10:
ProductionDataError_IndoPrint2:= CONCAT(ProductionData_IndoPrintError11.SERIALNOERROR,',');
ProductionDataError_IndoPrint2:=	 CONCAT( ProductionDataError_IndoPrint2,ProductionData_IndoPrintError11.SDATEERROR	);
ProductionDataError_IndoPrint2:= CONCAT( ProductionDataError_IndoPrint2,',');
(*ProductionDataError_IndoPrint2:=	 CONCAT( ProductionDataError_IndoPrint2,ProductionData_IndoPrintError11.STIMEEROOR);
ProductionDataError_IndoPrint2:= CONCAT( ProductionDataError_IndoPrint2,',');
ProductionDataError_IndoPrint2:=	 CONCAT( ProductionDataError_IndoPrint2,ProductionData_IndoPrintError11.SHIFTERROR	);
ProductionDataError_IndoPrint2:= CONCAT( ProductionDataError_IndoPrint2,',');*)
ProductionDataError_IndoPrint2:=	 CONCAT( ProductionDataError_IndoPrint2,ProductionData_IndoPrintError11.ERRORIDERROR);
ProductionDataError_IndoPrint2:= CONCAT( ProductionDataError_IndoPrint2,'$0A');
(*ProductionData_IndoPrint2:=	 CONCAT( ProductionData_IndoPrint2,ProductionData_IndoPrint11.LOTNO);
ProductionData_IndoPrint2:= CONCAT( ProductionData_IndoPrint2,',');
ProductionData_IndoPrint2:=	 CONCAT( ProductionData_IndoPrint2,ProductionData_IndoPrint11.DFLTNETWEIGHT);
ProductionData_IndoPrint2:= CONCAT( ProductionData_IndoPrint2,',');
ProductionData_IndoPrint2:=	 CONCAT( ProductionData_IndoPrint2,ProductionData_IndoPrint11.ACTNETWEIGHT);
ProductionData_IndoPrint2:= CONCAT( ProductionData_IndoPrint2,'$0A');
ProductionData_IndoPrint2:=	 CONCAT( ProductionData_IndoPrint2,ProductionData_IndoPrint11.DFLTGROSSWEIGHT);
ProductionData_IndoPrint2:= CONCAT( ProductionData_IndoPrint2,',');
ProductionData_IndoPrint2:=	 CONCAT( ProductionData_IndoPrint2,ProductionData_IndoPrint11.ACTGROSSWEIGHT);
ProductionData_IndoPrint2:= CONCAT( ProductionData_IndoPrint2,'$0A');
ProductionData_IndoPrint2:=	 CONCAT( ProductionData_IndoPrint2,ProductionData_IndoPrint11.NetWt9);
ProductionData_IndoPrint2:= CONCAT( ProductionData_IndoPrint2,',');
ProductionData_IndoPrint2:=	 CONCAT( ProductionData_IndoPrint2,ProductionData_IndoPrint11.NetWt10);
ProductionData_IndoPrint2:= CONCAT( ProductionData_IndoPrint2,',');
ProductionData_IndoPrint2:=	 CONCAT( ProductionData_IndoPrint2,ProductionData_IndoPrint11.NetWt11);
ProductionData_IndoPrint2:= CONCAT( ProductionData_IndoPrint2,',');
ProductionData_IndoPrint2:=	 CONCAT( ProductionData_IndoPrint2,ProductionData_IndoPrint11.NetWt12);
ProductionData_IndoPrint2:= CONCAT( ProductionData_IndoPrint2,',');*)
ReportBot1Error_Indo:=FALSE;ReportSaveErrror:=FALSE;
IndoReport:=15;


11:	ProductionDataValuesError_IndoPrint_Com:=ProductionDataError_IndoPrint2;
TON_Indo3(IN:=TRUE , PT:=t#5s , Q=> , ET=> );
	FB_FileWrite_Indo.bExecute:=TRUE;
	IF NOT FB_FileWrite_Indo.bBusy AND NOT FB_FileWrite_Indo.bError AND TON_Indo3.Q THEN IndoReport:=IndoReport+1; END_IF

12:	FB_FileWrite_Indo.bExecute:=FALSE;(*ProductionData_IndoPrint:='';*)IndoReport:=IndoReport+1;

13:	ReportBot2Error_Indo:=TRUE;
	IF ReportBot2Error_Indo THEN IndoReport:=IndoReport+1;END_IF

14:(*	ProductionData_IndoPrint2:= CONCAT(ProductionData_IndoPrint11.NetWt13,',');
ProductionData_IndoPrint2:=	 CONCAT( ProductionData_IndoPrint2,ProductionData_IndoPrint11.NetWt14	);
ProductionData_IndoPrint2:= CONCAT( ProductionData_IndoPrint2,',');
ProductionData_IndoPrint2:=	 CONCAT( ProductionData_IndoPrint2,ProductionData_IndoPrint11.NetWt15);
ProductionData_IndoPrint2:= CONCAT( ProductionData_IndoPrint2,',');
ProductionData_IndoPrint2:=	 CONCAT( ProductionData_IndoPrint2,ProductionData_IndoPrint11.NetWt16);
ProductionData_IndoPrint2:= CONCAT( ProductionData_IndoPrint2,',');
ProductionData_IndoPrint2:=	 CONCAT( ProductionData_IndoPrint2,ProductionData_IndoPrint11.NetWt17);
ProductionData_IndoPrint2:= CONCAT( ProductionData_IndoPrint2,',');
ProductionData_IndoPrint2:=	 CONCAT( ProductionData_IndoPrint2,ProductionData_IndoPrint11.NetWt18);
ProductionData_IndoPrint2:= CONCAT( ProductionData_IndoPrint2,',');
ProductionData_IndoPrint2:=	 CONCAT( ProductionData_IndoPrint2,ProductionData_IndoPrint11.NetWt19);
ProductionData_IndoPrint2:= CONCAT( ProductionData_IndoPrint2,',');
ProductionData_IndoPrint2:=	 CONCAT( ProductionData_IndoPrint2,ProductionData_IndoPrint11.NetWt20);
ProductionData_IndoPrint2:= CONCAT( ProductionData_IndoPrint2,',');
ProductionData_IndoPrint2:=	 CONCAT( ProductionData_IndoPrint2,ProductionData_IndoPrint11.NetWt21);
ProductionData_IndoPrint2:= CONCAT( ProductionData_IndoPrint2,',');
ProductionData_IndoPrint2:=	 CONCAT( ProductionData_IndoPrint2,ProductionData_IndoPrint11.NetWt22);
ProductionData_IndoPrint2:= CONCAT( ProductionData_IndoPrint2,',');
ProductionData_IndoPrint2:=	 CONCAT( ProductionData_IndoPrint2,ProductionData_IndoPrint11.NetWt23);
ProductionData_IndoPrint2:= CONCAT( ProductionData_IndoPrint2,',');
ProductionData_IndoPrint2:=	 CONCAT( ProductionData_IndoPrint2,ProductionData_IndoPrint11.NetWt24);
ProductionData_IndoPrint2:= CONCAT( ProductionData_IndoPrint2,'$0A');*)
ReportBot2Error_Indo:=FALSE;
IndoReport:=IndoReport+1;

15:ProductionDataValuesError_IndoPrint_Com:=ProductionDataError_IndoPrint2;
TON_Indo4(IN:=TRUE , PT:=t#5s , Q=> , ET=> );

	FB_FileWrite_Indo.bExecute:=TRUE; IndoReport:=IndoReport+1;
	(*IF NOT FB_FileWrite_Indo.bBusy AND NOT FB_FileWrite_Indo.bError AND TON_Indo4.Q  THEN IndoReport:=IndoReport+1;END_IF*)

16:	IF NOT FB_FileWrite_Indo.bBusy AND NOT FB_FileWrite_Indo.bError (*AND TON_Indo4.Q*)  THEN FB_FileWrite_Indo.bExecute:=FALSE; IndoReport:=IndoReport+1;END_IF


17:	TON_Indo3(IN:=FALSE);TON_Indo4(IN:=FALSE);TON_Indo2(IN:=FALSE);TON_Indo1(IN:=FALSE);FB_FileWrite_Indo.bExecute:=FALSE;IndoReport:=IndoReport+1;

18:	FB_FileClose_Indo.bExecute:=TRUE;
	 IF NOT FB_FileClose_Indo.bBusy AND NOT FB_FileClose_Indo.bError THEN  IndoReport:=20;END_IF

19:	IF bANewDayError THEN IndoReport:=IndoReport+1;
	ELSIF NOT bANewDayError THEN FB_FileOpen_Indo.bExecute:=FALSE; IndoReport:=9;
END_IF

20:	FB_FileOpen_Indo.bExecute:=FALSE;SerialNoError:=SerialNoError+1;IndoReport:=9;

END_CASE

R_TRIG_ErrorRepo_Int(CLK:=bInitializeHmi , Q=> );

IF sDay <> sOldDayError THEN bANewDayError:=TRUE;IndoReport:=0; END_IF
TON_NEWDAYError(IN:=bANewDayError , PT:=T#0.5s , Q=> , ET=> );



CASE WriteError OF
0:	IF FB_FileWrite_Indo.bError THEN FB_FileWrite_Indo.bExecute:=FALSE;TON_writedly(IN:=FALSE);
	WriteError:=WriteError+1;END_IF

1:	TON_writedly(IN:=TRUE , PT:=t#2s , Q=> , ET=> );
	IF TON_writedly.Q THEN FB_FileWrite_Indo.bExecute:=TRUE;WriteError:=WriteError+1;END_IF

2:	TON_writedly(IN:=FALSE);WriteError:=0;

END_CASE




CASE OpenError OF


0:	IF FB_FileWrite_Indo.bError THEN FB_FileWrite_Indo.bExecute:=FALSE;TON_Opendly(IN:=FALSE);
	OpenError:=OpenError+1;END_IF

1:	TON_Opendly(IN:=TRUE , PT:=t#2s , Q=> , ET=> );
	IF TON_Opendly.Q THEN FB_FileWrite_Indo.bExecute:=TRUE;OpenError:=OpenError+1;END_IF

2:	TON_Opendly(IN:=FALSE);OpenError:=0;

END_CASE









		ProductionData_IndoPrintError11.SERIALNOERROR	:=DINT_TO_STRING(SerialNoError);
		ProductionData_IndoPrintError11.SDATEERROR	:=(sTIME);
		(*ProductionData_IndoPrintError11.SHIFTERROR	:=(sShitToReport);*)
		ProductionData_IndoPrintError11.ERRORIDERROR	:=(AlarmData);
		(*ProductionData_IndoPrint11.LOTNO	:=(LOTNO_DIS);
		ProductionData_IndoPrint11.DFLTNETWEIGHT	:=(Default_NetWeight_Report);
		ProductionData_IndoPrint11.ACTNETWEIGHT	:=(Actual_NetWeight_Report);
		ProductionData_IndoPrint11.DFLTGROSSWEIGHT	:=(Default_GrossWeight_Report);
		ProductionData_IndoPrint11.ACTGROSSWEIGHT	:=(Actual_GrossWeight_Report);
		ProductionData_IndoPrint11.NetWt9	:=REAL_TO_STRING(Cone_9_Wt);
		ProductionData_IndoPrint11.NetWt10	:=REAL_TO_STRING(Cone_10_Wt);
		ProductionData_IndoPrint11.NetWt11	:=REAL_TO_STRING(Cone_11_Wt);
		ProductionData_IndoPrint11.NetWt12	:=REAL_TO_STRING(Cone_12_Wt);
		ProductionData_IndoPrint11.NetWt13	:=REAL_TO_STRING(Cone_13_Wt);
		ProductionData_IndoPrint11.NetWt14	:=REAL_TO_STRING(Cone_14_Wt);
		ProductionData_IndoPrint11.NetWt15	:=REAL_TO_STRING(Cone_15_Wt);
		ProductionData_IndoPrint11.NetWt16	:=REAL_TO_STRING(Cone_16_Wt);
		ProductionData_IndoPrint11.NetWt17	:=REAL_TO_STRING(Cone_17_Wt);
		ProductionData_IndoPrint11.NetWt18	:=REAL_TO_STRING(Cone_18_Wt);
		ProductionData_IndoPrint11.NetWt19	:=REAL_TO_STRING(Cone_19_Wt);
		ProductionData_IndoPrint11.NetWt20	:=REAL_TO_STRING(Cone_20_Wt);
		ProductionData_IndoPrint11.NetWt21	:=REAL_TO_STRING(Cone_21_Wt);
		ProductionData_IndoPrint11.NetWt22	:=REAL_TO_STRING(Cone_22_Wt);
		ProductionData_IndoPrint11.NetWt23	:=REAL_TO_STRING(Cone_23_Wt);
		ProductionData_IndoPrint11.NetWt24	:=REAL_TO_STRING(Cone_24_Wt);*)
END_PROGRAM

(* POU Date_Time, ST *)
PROGRAM Date_Time
VAR
	ReportPath: STRING;



	sDayF1: STRING;
	sMonthF1: STRING;
	sDayMonth1: STRING;

END_VAR
				(****************REPORT DATA***********)
IF DfltWtPrint THEN NetwtPrint:=Default_NetWeight_Report;
ELSIF NOT DfltWtPrint THEN NetwtPrint:=Actual_NetWeight_Report;END_IF

IF GrossWtPrintDflt THEN GrosswtPrint:=Default_GrossWeight_Report;
ELSE GrosswtPrint:=Actual_GrossWeight_Report;END_IF



Actual_NetWeight_Report:=MID(STR:=REAL_TO_STRING(var_5), LEN:=6, POS:=1);
Default_NetWeight_Report:=MID(STR:=REAL_TO_STRING(DefaultNetWt), LEN:=6, POS:=1);

Actual_GrossWeight_Report:=MID(STR:=REAL_TO_STRING(rGrossWeight), LEN:=6, POS:=1);
Default_GrossWeight_Report:=MID(STR:=REAL_TO_STRING(DefaultGrossWt), LEN:=6, POS:=1);




					(****************DATE AND TIME***********)

(*======================= RTC==============================*)

FB_DateTime_1(NET_ID:='5.69.203.190.1.1 ' , Date_Time=> );

IF FB_DateTime_1.FBLTIME.systemTime.wHour >0 AND  FB_DateTime_1.FBLTIME.systemTime.wHour<9 THEN sHourPreFix:='0';

sHou:=CONCAT(STR1:=sHourPreFix, Str2:=WORD_TO_STRING(FB_DateTime_1.FBLTIME.systemTime.wHour));

ELSIF FB_DateTime_1.FBLTIME.systemTime.wHour >=10 AND  FB_DateTime_1.FBLTIME.systemTime.wHour<=24 THEN

sHou:=WORD_TO_STRING(FB_DateTime_1.FBLTIME.systemTime.wHour);

END_IF




IF FB_DateTime_1.FBLTIME.systemTime.wDay >0 AND  FB_DateTime_1.FBLTIME.systemTime.wDay<10 THEN sDayPreFix:='0';

sDay:=CONCAT(STR1:=sDayPreFix, Str2:=WORD_TO_STRING(FB_DateTime_1.FBLTIME.systemTime.wDay));

ELSIF FB_DateTime_1.FBLTIME.systemTime.wDay >=10 AND  FB_DateTime_1.FBLTIME.systemTime.wDay<=31 THEN

sDay:=WORD_TO_STRING(FB_DateTime_1.FBLTIME.systemTime.wDay);

END_IF




IF FB_DateTime_1.FBLTIME.systemTime.wMonth >0 AND  FB_DateTime_1.FBLTIME.systemTime.wMonth<10 THEN sMonthPreFix:='0';

sMonth:=CONCAT(STR1:=sMonthPreFix, Str2:=WORD_TO_STRING(FB_DateTime_1.FBLTIME.systemTime.wMonth));

ELSIF FB_DateTime_1.FBLTIME.systemTime.wMonth >=10 AND  FB_DateTime_1.FBLTIME.systemTime.wMonth<=12 THEN

sMonth:=WORD_TO_STRING(FB_DateTime_1.FBLTIME.systemTime.wMonth);

END_IF



sDayF1:=CONCAT(STR1:=sDay, STR2:=':');
sMonthF1:=CONCAT(STR1:=sMonth, STR2:=':');
sDayMonth1:=CONCAT(STR1:=sDayF1, STR2:=sMonthF1);
sDayMonthYear1:=CONCAT(STR1:=sDayMonth1, STR2:=WORD_TO_STRING(FB_DateTime_1.FBLTIME.systemTime.wYear));


sDaateReport:=(sDayMonthYear1);





sDayF:=CONCAT(STR1:=sDay, STR2:='_');
sMonthF:=CONCAT(STR1:=sMonth, STR2:='_');
sDayMonth:=CONCAT(STR1:=sDayF, STR2:=sMonthF);
sDayMonthYear:=CONCAT(STR1:=sDayMonth, STR2:=WORD_TO_STRING(FB_DateTime_1.FBLTIME.systemTime.wYear));

ReportPath:=CONCAT(STR1:='ProductionData', STR2:='_');
ReportPath_Final:=CONCAT(STR1:=ReportPath, STR2:=sDayMonthYear);

ReportPath_Final_1:=CONCAT(STR1:='\\ACP\Reports\', STR2:=ReportPath_Final);
ReportPath_Final_2:=CONCAT(STR1:=ReportPath_Final_1, STR2:='.csv');





sDayF1:=CONCAT(STR1:=sDay, STR2:=':');
sMonthF1:=CONCAT(STR1:=sMonth, STR2:=':');
sDayMonth1:=CONCAT(STR1:=sDayF1, STR2:=sMonthF1);
sDayMonthYear1:=CONCAT(STR1:=sDayMonth1, STR2:=WORD_TO_STRING(FB_DateTime_1.FBLTIME.systemTime.wYear));


sDaateReport:=(sDayMonthYear1);





sDayF:=CONCAT(STR1:=sDay, STR2:='_');
sMonthF:=CONCAT(STR1:=sMonth, STR2:='_');
sDayMonth:=CONCAT(STR1:=sDayF, STR2:=sMonthF);
sDayMonthYear:=CONCAT(STR1:=sDayMonth, STR2:=WORD_TO_STRING(FB_DateTime_1.FBLTIME.systemTime.wYear));

ReportPathError:=CONCAT(STR1:='ErrorData', STR2:='_');
ReportPath_FinalError:=CONCAT(STR1:=ReportPathError, STR2:=sDayMonthYear);

ReportPath_Final_1Error:=CONCAT(STR1:='\\ACP\Reports\', STR2:=ReportPath_FinalError);
ReportPath_Final_2Error:=CONCAT(STR1:=ReportPath_Final_1Error, STR2:='.csv');








DateTimeVar:=FB_DateTime_1.Date_Time;
END_PROGRAM

(* POU Parameters, ST *)
PROGRAM Parameters
VAR
	R_TRIG_1: R_TRIG;

	PrintVar: INT;




	ItemCodeHm21: BOOL;
END_VAR
IF SAVE AND PRGNO=1 AND NegTolEnableHmi THEN NegTol1:=1;ELSIF SAVE AND PRGNO=1 AND NOT  NegTolEnableHmi THEN  NegTol1:=0;END_IF
IF SAVE AND PRGNO=2 AND NegTolEnableHmi THEN NegTol2:=1;ELSIF SAVE AND PRGNO=2 AND NOT NegTolEnableHmi THEN  NegTol2:=0;END_IF
IF SAVE AND PRGNO=3 AND NegTolEnableHmi THEN NegTol3:=1;ELSIF SAVE AND PRGNO=3 AND NOT NegTolEnableHmi THEN  NegTol3:=0;END_IF
IF SAVE AND PRGNO=4 AND NegTolEnableHmi THEN NegTol4:=1;ELSIF SAVE AND PRGNO=4 AND NOT NegTolEnableHmi THEN  NegTol4:=0;END_IF
IF SAVE AND PRGNO=5 AND NegTolEnableHmi THEN NegTol5:=1;ELSIF SAVE AND PRGNO=5 AND NOT NegTolEnableHmi THEN  NegTol5:=0;END_IF

IF SAVE AND PRGNO=1 THEN

	PRGNO1:=PRGNO;
	COUNT1:=COUNT;
	CARTONNO1:=CARTONNO;
	DFLTNETWT1:=DFLTNETWT;
	DFLTGROSSWT1:=DFLTGROSSWT;
	BLEND1:=BLEND;
	SHADE1:=SHADE;
	CONETIP1:=CONETIP;
	CONELENGTH1:=CONELENGTH;
	CONENETWT1:=CONENETWT;
	NOOFCONES1:=NOOFCONES;
	LOTNO1:=LOTNO;
	WORKORDERNO1:=WORKORDERNO;
	NETWTTOL1:=NETWTTOL;
	GROSSWTTOL1:=GROSSWTTOL;
	DOM_EXPORT1:=DOM_EXPORT;
	PACKTYPE1:=PACKTYPE;

	ItemCodeHmi1:=ItemCodeHmi;
	IssueDesp1:=IssueDesp;
	Location1:=Location;
	Description1:=Description;
	Remarks1:=Remarks;
	Fyear1:=Fyear;
	AvgCount1:=AvgCount;
	TareWeight1:=TareWeight;
	BarCode1:=BarCode;
	WorkFlag1:=WorkFlag;
	EmptyConeWt1:=EmptyConeWt;


ELSIF SAVE AND PRGNO=2 THEN

	PRGNO2:=PRGNO;
	COUNT2:=COUNT;
	CARTONNO2:=CARTONNO;
	DFLTNETWT2:=DFLTNETWT;
	DFLTGROSSWT2:=DFLTGROSSWT;
	BLEND2:=BLEND;
	SHADE2:=SHADE;
	CONETIP2:=CONETIP;
	CONELENGTH2:=CONELENGTH;
	CONENETWT2:=CONENETWT;
	NOOFCONES2:=NOOFCONES;
	LOTNO2:=LOTNO;
	WORKORDERNO2:=WORKORDERNO;
	NETWTTOL2:=NETWTTOL;
	GROSSWTTOL2:=GROSSWTTOL;
	DOM_EXPORT2:=DOM_EXPORT;
	PACKTYPE2:=PACKTYPE;

	ItemCodeHmI2:=ItemCodeHmi;
	IssueDesp2:=IssueDesp;
	Location2:=Location;
	Description2:=Description;
	Remarks2:=Remarks;
	Fyear2:=Fyear;
	AvgCount2:=AvgCount;
	TareWeight2:=TareWeight;
	BarCode2:=BarCode;
	WorkFlag2:=WorkFlag;
	EmptyConeWt2:=EmptyConeWt;

ELSIF SAVE AND PRGNO=3 THEN

	PRGNO3:=PRGNO;
	COUNT3:=COUNT;
	CARTONNO3:=CARTONNO;
	DFLTNETWT3:=DFLTNETWT;
	DFLTGROSSWT3:=DFLTGROSSWT;
	BLEND3:=BLEND;
	SHADE3:=SHADE;
	CONETIP3:=CONETIP;
	CONELENGTH3:=CONELENGTH;
	CONENETWT3:=CONENETWT;
	NOOFCONES3:=NOOFCONES;
	LOTNO3:=LOTNO;
	WORKORDERNO3:=WORKORDERNO;
	NETWTTOL3:=NETWTTOL;
	GROSSWTTOL3:=GROSSWTTOL;
	DOM_EXPORT3:=DOM_EXPORT;
	PACKTYPE3:=PACKTYPE;

ItemCodeHmI3:=ItemCodeHmi;
	IssueDesp3:=IssueDesp;
	Location3:=Location;
	Description3:=Description;
	Remarks3:=Remarks;
	Fyear3:=Fyear;
	AvgCount3:=AvgCount;
	TareWeight3:=TareWeight;
	BarCode3:=BarCode;
	WorkFlag3:=WorkFlag;
	EmptyConeWt3:=EmptyConeWt;


ELSIF SAVE AND PRGNO=4 THEN

	PRGNO4:=PRGNO;
	COUNT4:=COUNT;
	CARTONNO4:=CARTONNO;
	DFLTNETWT4:=DFLTNETWT;
	DFLTGROSSWT4:=DFLTGROSSWT;
	BLEND4:=BLEND;
	SHADE4:=SHADE;
	CONETIP4:=CONETIP;
	CONELENGTH4:=CONELENGTH;
	CONENETWT4:=CONENETWT;
	NOOFCONES4:=NOOFCONES;
	LOTNO4:=LOTNO;
	WORKORDERNO4:=WORKORDERNO;
	NETWTTOL4:=NETWTTOL;
	GROSSWTTOL4:=GROSSWTTOL;
	DOM_EXPORT4:=DOM_EXPORT;
	PACKTYPE4:=PACKTYPE;

ItemCodeHmI4:=ItemCodeHmi;
	IssueDesp4:=IssueDesp;
	Location4:=Location;
	Description4:=Description;
	Remarks4:=Remarks;
	Fyear4:=Fyear;
	AvgCount4:=AvgCount;
	TareWeight4:=TareWeight;
	BarCode4:=BarCode;
	WorkFlag4:=WorkFlag;
	EmptyConeWt4:=EmptyConeWt;

ELSIF SAVE AND PRGNO=5 THEN

	PRGNO5:=PRGNO;
	COUNT5:=COUNT;
	CARTONNO5:=CARTONNO;
	DFLTNETWT5:=DFLTNETWT;
	DFLTGROSSWT5:=DFLTGROSSWT;
	BLEND5:=BLEND;
	SHADE5:=SHADE;
	CONETIP5:=CONETIP;
	CONELENGTH5:=CONELENGTH;
	CONENETWT5:=CONENETWT;
	NOOFCONES5:=NOOFCONES;
	LOTNO5:=LOTNO;
	WORKORDERNO5:=WORKORDERNO;
	NETWTTOL5:=NETWTTOL;
	GROSSWTTOL5:=GROSSWTTOL;
	DOM_EXPORT5:=DOM_EXPORT;
	PACKTYPE5:=PACKTYPE;

	ItemCodeHmI5:=ItemCodeHmi;
	IssueDesp5:=IssueDesp;
	Location5:=Location;
	Description5:=Description;
	Remarks5:=Remarks;
	Fyear5:=Fyear;
	AvgCount5:=AvgCount;
	TareWeight5:=TareWeight;
	BarCode5:=BarCode;
	WorkFlag5:=WorkFlag;
	EmptyConeWt5:=EmptyConeWt;

ELSIF SAVE AND PRGNO=6 THEN

	PRGNO6:=PRGNO;
	COUNT6:=COUNT;
	DETAILS6:=DETAILS;
	LOTNO6:=LOTNO;
	CARTONNO6:=CARTONNO;
	WORKORDERNO6:=WORKORDERNO;
	BLEND6:=BLEND;
	SHADE6:=SHADE;
	CONETIP6:=CONETIP;
	CONELENGTH6:=CONELENGTH;
	CONENETWT6:=CONENETWT;
	DFLTNETWT6:=DFLTNETWT;
	NETWTTOL6:=NETWTTOL;
	DFLTGROSSWT6:=DFLTGROSSWT;
	GROSSWTTOL6:=GROSSWTTOL;


ELSIF SAVE AND PRGNO=7 THEN

	PRGNO7:=PRGNO;
	COUNT7:=COUNT;
	DETAILS7:=DETAILS;
	LOTNO7:=LOTNO;
	CARTONNO7:=CARTONNO;
	WORKORDERNO7:=WORKORDERNO;
	BLEND7:=BLEND;
	SHADE7:=SHADE;
	CONETIP7:=CONETIP;
	CONELENGTH7:=CONELENGTH;
	CONENETWT7:=CONENETWT;
	DFLTNETWT7:=DFLTNETWT;
	NETWTTOL7:=NETWTTOL;
	DFLTGROSSWT7:=DFLTGROSSWT;
	GROSSWTTOL7:=GROSSWTTOL;


ELSIF SAVE AND PRGNO=8 THEN

	PRGNO8:=PRGNO;
	COUNT8:=COUNT;
	DETAILS8:=DETAILS;
	LOTNO8:=LOTNO;
	CARTONNO8:=CARTONNO;
	WORKORDERNO8:=WORKORDERNO;
	BLEND8:=BLEND;
	SHADE8:=SHADE;
	CONETIP8:=CONETIP;
	CONELENGTH8:=CONELENGTH;
	CONENETWT8:=CONENETWT;
	DFLTNETWT8:=DFLTNETWT;
	NETWTTOL8:=NETWTTOL;
	DFLTGROSSWT8:=DFLTGROSSWT;
	GROSSWTTOL8:=GROSSWTTOL;


ELSIF SAVE AND PRGNO=9 THEN

	PRGNO9:=PRGNO;
	COUNT9:=COUNT;
	DETAILS9:=DETAILS;
	LOTNO9:=LOTNO;
	CARTONNO9:=CARTONNO;
	WORKORDERNO9 :=WORKORDERNO;
	BLEND9 :=BLEND;
	SHADE9 :=SHADE;
	CONETIP9 :=CONETIP;
	CONELENGTH9 :=CONELENGTH;
	CONENETWT9 :=CONENETWT;
	DFLTNETWT9 :=DFLTNETWT;
	NETWTTOL9 :=NETWTTOL;
	DFLTGROSSWT9 :=DFLTGROSSWT;
	GROSSWTTOL9 :=GROSSWTTOL;


ELSIF SAVE AND PRGNO=10 THEN

	PRGNO10:=PRGNO;
	COUNT10:=COUNT;
	DETAILS10:=DETAILS;
	LOTNO10:=LOTNO;
	CARTONNO10:=CARTONNO;
	WORKORDERNO10:=WORKORDERNO;
	BLEND10:=BLEND;
	SHADE10:=SHADE;
	CONETIP10:=CONETIP;
	CONELENGTH10:=CONELENGTH;
	CONENETWT10:=CONENETWT;
	DFLTNETWT10:=DFLTNETWT;
	NETWTTOL10:=NETWTTOL;
	DFLTGROSSWT10:=DFLTGROSSWT;
	GROSSWTTOL10:=GROSSWTTOL;

END_IF










IF LOAD AND PRGNO_LOAD=1 THEN


	PRGNO_DIS:=PRGNO1;
	COUNT_DIS:=COUNT1;
	CARTONNO_DIS:=CARTONNO1;
	DFLTNETWT_DIS:=DFLTNETWT1;
	DFLTGROSSWT_DIS:=DFLTGROSSWT1;
	BLEND_DIS:=BLEND1;
	SHADE_DIS:=SHADE1;
	CONETIP_DIS:=CONETIP1;
	CONELENGTH_DIS:=CONELENGTH1;
	CONENETWT_DIS:=CONENETWT1;
	NOOFCONES_DIS:=NOOFCONES1;
	LOTNO_DIS:=LOTNO1;
	WORKORDERNO_DIS:=WORKORDERNO1;
	NETWTTOL_DIS:=NETWTTOL1;
	GROSSWTTOL_DIS:=GROSSWTTOL1;
	DOM_EXPORT_DIS:=DOM_EXPORT1;
	PACKTYPE_DIS:=PACKTYPE1;
	NegTol_DIS:=NegTol1;
	PRG1RUNNING:=TRUE;
	PRG2RUNNING:=FALSE;
	PRG3RUNNING:=FALSE;
	PRG4RUNNING:=FALSE;
	PRG5RUNNING:=FALSE;
	PRG6RUNNING:=FALSE;
	PRG7RUNNING:=FALSE;
	PRG8RUNNING:=FALSE;
	PRG9RUNNING:=FALSE;
	PRG10RUNNING:=FALSE;


ItemCodeHmi_DIS:=ItemCodeHmi1;
IssueDesp_DIS:=	IssueDesp1;
Location_DIS:=Location1;
Description_DIS:=	Description1;
Remarks_DIS:=	Remarks1;
Fyear_DIS:=	Fyear1;
AvgCount_DIS:=	AvgCount1;
TareWeight_DIS:=	TareWeight1;
BarCode_DIS:=	BarCode1;
WorkFlag_DIS:=	WorkFlag1;
EmptyConeWt_DIS:=EmptyConeWt1;

ELSIF LOAD AND PRGNO_LOAD=2 THEN

	PRGNO_DIS:=PRGNO2;
	COUNT_DIS:=COUNT2;
	CARTONNO_DIS:=CARTONNO2;
	DFLTNETWT_DIS:=DFLTNETWT2;
	DFLTGROSSWT_DIS:=DFLTGROSSWT2;
	BLEND_DIS:=BLEND2;
	SHADE_DIS:=SHADE2;
	CONETIP_DIS:=CONETIP2;
	CONELENGTH_DIS:=CONELENGTH2;
	CONENETWT_DIS:=CONENETWT2;
	NOOFCONES_DIS:=NOOFCONES2;
	LOTNO_DIS:=LOTNO2;
	WORKORDERNO_DIS:=WORKORDERNO2;
	NETWTTOL_DIS:=NETWTTOL2;
	GROSSWTTOL_DIS:=GROSSWTTOL2;
	DOM_EXPORT_DIS:=DOM_EXPORT2;
	PACKTYPE_DIS:=PACKTYPE2;
	NegTol_DIS:=NegTol2;
	PRG2RUNNING:=TRUE;
	PRG1RUNNING:=FALSE;
	PRG3RUNNING:=FALSE;
	PRG4RUNNING:=FALSE;
	PRG5RUNNING:=FALSE;
	PRG6RUNNING:=FALSE;
	PRG7RUNNING:=FALSE;
	PRG8RUNNING:=FALSE;
	PRG9RUNNING:=FALSE;
	PRG10RUNNING:=FALSE;


ItemCodeHmi_DIS:=ItemCodeHmi2;
IssueDesp_DIS:=	IssueDesp2;
Location_DIS:=Location2;
Description_DIS:=	Description2;
Remarks_DIS:=	Remarks2;
Fyear_DIS:=	Fyear2;
AvgCount_DIS:=	AvgCount2;
TareWeight_DIS:=	TareWeight2;
BarCode_DIS:=	BarCode2;
WorkFlag_DIS:=	WorkFlag2;
EmptyConeWt_DIS:=EmptyConeWt2;

ELSIF LOAD AND PRGNO_LOAD=3 THEN

	PRGNO_DIS:=PRGNO3;
	COUNT_DIS:=COUNT3;
	CARTONNO_DIS:=CARTONNO3;
	DFLTNETWT_DIS:=DFLTNETWT3;
	DFLTGROSSWT_DIS:=DFLTGROSSWT3;
	BLEND_DIS:=BLEND3;
	SHADE_DIS:=SHADE3;
	CONETIP_DIS:=CONETIP3;
	CONELENGTH_DIS:=CONELENGTH3;
	CONENETWT_DIS:=CONENETWT3;
	NOOFCONES_DIS:=NOOFCONES3;
	LOTNO_DIS:=LOTNO3;
	WORKORDERNO_DIS:=WORKORDERNO3;
	NETWTTOL_DIS:=NETWTTOL3;
	GROSSWTTOL_DIS:=GROSSWTTOL3;
	DOM_EXPORT_DIS:=DOM_EXPORT3;
	PACKTYPE_DIS:=PACKTYPE3;
	NegTol_DIS:=NegTol3;
	PRG3RUNNING:=TRUE;
	PRG2RUNNING:=FALSE;
	PRG1RUNNING:=FALSE;
	PRG4RUNNING:=FALSE;
	PRG5RUNNING:=FALSE;
	PRG6RUNNING:=FALSE;
	PRG7RUNNING:=FALSE;
	PRG8RUNNING:=FALSE;
	PRG9RUNNING:=FALSE;
	PRG10RUNNING:=FALSE;


ItemCodeHmi_DIS:=ItemCodeHmi3;
IssueDesp_DIS:=	IssueDesp3;
Location_DIS:=Location3;
Description_DIS:=	Description3;
Remarks_DIS:=	Remarks3;
Fyear_DIS:=	Fyear3;
AvgCount_DIS:=	AvgCount3;
TareWeight_DIS:=	TareWeight3;
BarCode_DIS:=	BarCode3;
WorkFlag_DIS:=	WorkFlag3;
EmptyConeWt_DIS:=EmptyConeWt3;


ELSIF LOAD AND PRGNO_LOAD=4 THEN

	PRGNO_DIS:=PRGNO4;
	COUNT_DIS:=COUNT4;
	CARTONNO_DIS:=CARTONNO4;
	DFLTNETWT_DIS:=DFLTNETWT4;
	DFLTGROSSWT_DIS:=DFLTGROSSWT4;
	BLEND_DIS:=BLEND4;
	SHADE_DIS:=SHADE4;
	CONETIP_DIS:=CONETIP4;
	CONELENGTH_DIS:=CONELENGTH4;
	CONENETWT_DIS:=CONENETWT4;
	NOOFCONES_DIS:=NOOFCONES4;
	LOTNO_DIS:=LOTNO4;
	WORKORDERNO_DIS:=WORKORDERNO4;
	NETWTTOL_DIS:=NETWTTOL4;
	GROSSWTTOL_DIS:=GROSSWTTOL4;
	DOM_EXPORT_DIS:=DOM_EXPORT4;
	PACKTYPE_DIS:=PACKTYPE4;
	NegTol_DIS:=NegTol4;
	PRG4RUNNING:=TRUE;
	PRG2RUNNING:=FALSE;
	PRG3RUNNING:=FALSE;
	PRG1RUNNING:=FALSE;
	PRG5RUNNING:=FALSE;
	PRG6RUNNING:=FALSE;
	PRG7RUNNING:=FALSE;
	PRG8RUNNING:=FALSE;
	PRG9RUNNING:=FALSE;
	PRG10RUNNING:=FALSE;



ItemCodeHmi_DIS:=ItemCodeHmi4;
IssueDesp_DIS:=	IssueDesp4;
Location_DIS:=Location4;
Description_DIS:=	Description4;
Remarks_DIS:=	Remarks4;
Fyear_DIS:=	Fyear4;
AvgCount_DIS:=	AvgCount4;
TareWeight_DIS:=	TareWeight4;
BarCode_DIS:=	BarCode4;
WorkFlag_DIS:=	WorkFlag4;
EmptyConeWt_DIS:=EmptyConeWt4;


ELSIF LOAD AND PRGNO_LOAD=5 THEN

	PRGNO_DIS:=PRGNO5;
	COUNT_DIS:=COUNT5;
	CARTONNO_DIS:=CARTONNO5;
	DFLTNETWT_DIS:=DFLTNETWT5;
	DFLTGROSSWT_DIS:=DFLTGROSSWT5;
	BLEND_DIS:=BLEND5;
	SHADE_DIS:=SHADE5;
	CONETIP_DIS:=CONETIP5;
	CONELENGTH_DIS:=CONELENGTH5;
	CONENETWT_DIS:=CONENETWT5;
	NOOFCONES_DIS:=NOOFCONES5;
	LOTNO_DIS:=LOTNO5;
	WORKORDERNO_DIS:=WORKORDERNO5;
	NETWTTOL_DIS:=NETWTTOL5;
	GROSSWTTOL_DIS:=GROSSWTTOL5;
	DOM_EXPORT_DIS:=DOM_EXPORT5;
	PACKTYPE_DIS:=PACKTYPE5;
	NegTol_DIS:=NegTol5;
	PRG5RUNNING:=TRUE;
	PRG2RUNNING:=FALSE;
	PRG3RUNNING:=FALSE;
	PRG4RUNNING:=FALSE;
	PRG1RUNNING:=FALSE;
	PRG6RUNNING:=FALSE;
	PRG7RUNNING:=FALSE;
	PRG8RUNNING:=FALSE;
	PRG9RUNNING:=FALSE;
	PRG10RUNNING:=FALSE;


ItemCodeHmi_DIS:=ItemCodeHmi5;
IssueDesp_DIS:=	IssueDesp5;
Location_DIS:=Location5;
Description_DIS:=	Description5;
Remarks_DIS:=	Remarks5;
Fyear_DIS:=	Fyear5;
AvgCount_DIS:=	AvgCount5;
TareWeight_DIS:=	TareWeight5;
BarCode_DIS:=	BarCode5;
WorkFlag_DIS:=	WorkFlag5;
EmptyConeWt_DIS:=EmptyConeWt5;

ELSIF LOAD AND PRGNO_LOAD=6 THEN

	PRGNO_DIS:=PRGNO6;
	COUNT_DIS:=COUNT6;
	DETAILS_DIS:=DETAILS6;
	LOTNO_DIS:=LOTNO6;
	CARTONNO_DIS:=CARTONNO6;
	WORKORDERNO_DIS:=WORKORDERNO6;
	BLEND_DIS:=BLEND6;
	SHADE_DIS:=SHADE6;
	CONETIP_DIS:=CONETIP6;
	CONELENGTH_DIS:=CONELENGTH6;
	CONENETWT_DIS:=CONENETWT6;
	DFLTNETWT_DIS:=DFLTNETWT6;
	NETWTTOL_DIS:=NETWTTOL6;
	DFLTGROSSWT_DIS:=DFLTGROSSWT6;
	GROSSWTTOL_DIS:=GROSSWTTOL6;
	PRG6RUNNING:=TRUE;
	PRG2RUNNING:=FALSE;
	PRG3RUNNING:=FALSE;
	PRG4RUNNING:=FALSE;
	PRG5RUNNING:=FALSE;
	PRG1RUNNING:=FALSE;
	PRG7RUNNING:=FALSE;
	PRG8RUNNING:=FALSE;
	PRG9RUNNING:=FALSE;
	PRG10RUNNING:=FALSE;

ELSIF LOAD AND PRGNO_LOAD=7 THEN

	PRGNO_DIS:=PRGNO7;
	COUNT_DIS:=COUNT7;
	DETAILS_DIS:=DETAILS7;
	LOTNO_DIS:=LOTNO7;
	CARTONNO_DIS:=CARTONNO7;
	WORKORDERNO_DIS:=WORKORDERNO7;
	BLEND_DIS:=BLEND7;
	SHADE_DIS:=SHADE7;
	CONETIP_DIS:=CONETIP7;
	CONELENGTH_DIS:=CONELENGTH7;
	CONENETWT_DIS:=CONENETWT7;
	DFLTNETWT_DIS:=DFLTNETWT7;
	NETWTTOL_DIS:=NETWTTOL7;
	DFLTGROSSWT_DIS:=DFLTGROSSWT7;
	GROSSWTTOL_DIS:=GROSSWTTOL7;
	PRG7RUNNING:=TRUE;
	PRG2RUNNING:=FALSE;
	PRG3RUNNING:=FALSE;
	PRG4RUNNING:=FALSE;
	PRG5RUNNING:=FALSE;
	PRG6RUNNING:=FALSE;
	PRG1RUNNING:=FALSE;
	PRG8RUNNING:=FALSE;
	PRG9RUNNING:=FALSE;
	PRG10RUNNING:=FALSE;


ELSIF LOAD AND PRGNO_LOAD=8 THEN

	PRGNO_DIS:=PRGNO8;
	COUNT_DIS:=COUNT8;
	DETAILS_DIS:=DETAILS8;
	LOTNO_DIS:=LOTNO8;
	CARTONNO_DIS:=CARTONNO8;
	WORKORDERNO_DIS:=WORKORDERNO8;
	BLEND_DIS:=BLEND8;
	SHADE_DIS:=SHADE8;
	CONETIP_DIS:=CONETIP8;
	CONELENGTH_DIS:=CONELENGTH8;
	CONENETWT_DIS:=CONENETWT8;
	DFLTNETWT_DIS:=DFLTNETWT8;
	NETWTTOL_DIS:=NETWTTOL8;
	DFLTGROSSWT_DIS:=DFLTGROSSWT8;
	GROSSWTTOL_DIS:=GROSSWTTOL8;
	PRG8RUNNING:=TRUE;
	PRG2RUNNING:=FALSE;
	PRG3RUNNING:=FALSE;
	PRG4RUNNING:=FALSE;
	PRG5RUNNING:=FALSE;
	PRG6RUNNING:=FALSE;
	PRG7RUNNING:=FALSE;
	PRG1RUNNING:=FALSE;
	PRG9RUNNING:=FALSE;
	PRG10RUNNING:=FALSE;


ELSIF LOAD AND PRGNO_LOAD=9 THEN

	PRGNO_DIS:=PRGNO9;
	COUNT_DIS:=COUNT9;
	DETAILS_DIS:=DETAILS9;
	LOTNO_DIS:=LOTNO9;
	CARTONNO_DIS:=CARTONNO9;
	WORKORDERNO_DIS:=WORKORDERNO9;
	BLEND_DIS:=BLEND9;
	SHADE_DIS:=SHADE9;
	CONETIP_DIS:=CONETIP9;
	CONELENGTH_DIS:=CONELENGTH9;
	CONENETWT_DIS:=CONENETWT9;
	DFLTNETWT_DIS:=DFLTNETWT9;
	NETWTTOL_DIS:=NETWTTOL9;
	DFLTGROSSWT_DIS:=DFLTGROSSWT9;
	GROSSWTTOL_DIS:=GROSSWTTOL9;
	PRG9RUNNING:=TRUE;
	PRG2RUNNING:=FALSE;
	PRG3RUNNING:=FALSE;
	PRG4RUNNING:=FALSE;
	PRG5RUNNING:=FALSE;
	PRG6RUNNING:=FALSE;
	PRG7RUNNING:=FALSE;
	PRG8RUNNING:=FALSE;
	PRG1RUNNING:=FALSE;
	PRG10RUNNING:=FALSE;


ELSIF LOAD AND PRGNO_LOAD=10 THEN

	PRGNO_DIS:=PRGNO10;
	COUNT_DIS:=COUNT10;
	DETAILS_DIS:=DETAILS10;
	LOTNO_DIS:=LOTNO10;
	CARTONNO_DIS:=CARTONNO10;
	WORKORDERNO_DIS:=WORKORDERNO10;
	BLEND_DIS:=BLEND10;
	SHADE_DIS:=SHADE10;
	CONETIP_DIS:=CONETIP10;
	CONELENGTH_DIS:=CONELENGTH10;
	CONENETWT_DIS:=CONENETWT10;
	DFLTNETWT_DIS:=DFLTNETWT10;
	NETWTTOL_DIS:=NETWTTOL10;
	DFLTGROSSWT_DIS:=DFLTGROSSWT10;
	GROSSWTTOL_DIS:=GROSSWTTOL10;
	PRG10RUNNING:=TRUE;
	PRG2RUNNING:=FALSE;
	PRG3RUNNING:=FALSE;
	PRG4RUNNING:=FALSE;
	PRG5RUNNING:=FALSE;
	PRG6RUNNING:=FALSE;
	PRG7RUNNING:=FALSE;
	PRG8RUNNING:=FALSE;
	PRG9RUNNING:=FALSE;
	PRG1RUNNING:=FALSE;

END_IF


IF PRG1RUNNING AND NegTol1=1 THEN negativetolerance1:=TRUE; ELSE negativetolerance1:=FALSE;END_IF

IF PRG2RUNNING AND NegTol2=1 THEN negativetolerance2:=TRUE; ELSE negativetolerance2:=FALSE;END_IF

IF PRG3RUNNING AND NegTol3=1 THEN negativetolerance3:=TRUE; ELSE negativetolerance3:=FALSE;END_IF

IF PRG4RUNNING AND NegTol4=1 THEN negativetolerance4:=TRUE; ELSE negativetolerance4:=FALSE;END_IF

IF PRG5RUNNING AND NegTol5=1 THEN negativetolerance5:=TRUE; ELSE negativetolerance5:=FALSE;END_IF

IF PRG1RUNNING AND negativetolerance1 THEN negativetolerance:=TRUE;
ELSIF PRG2RUNNING AND negativetolerance2 THEN negativetolerance:=TRUE;
ELSIF PRG3RUNNING AND negativetolerance3 THEN negativetolerance:=TRUE;
ELSIF PRG4RUNNING AND negativetolerance4 THEN negativetolerance:=TRUE;
ELSIF PRG5RUNNING AND negativetolerance5 THEN negativetolerance:=TRUE;END_IF
IF LOAD THEN negativetolerance:=FALSE;END_IF

R_TRIG_1(CLK:=(ReportPrint (*OR bABagComplete*)) , Q=> );



IF R_TRIG_1.Q THEN
CARTONNO_DIS:=CARTONNO_DIS+1;
ReportPrint:=FALSE;
ReportSave:=TRUE;
PrintOk:=TRUE;
END_IF

IF PRGNO_LOAD=3 AND R_TRIG_1.Q THEN CARTONNO3:=CARTONNO_DIS;
ELSIF PRGNO_LOAD=2 AND R_TRIG_1.Q THEN CARTONNO2:=CARTONNO_DIS;
ELSIF PRGNO_LOAD=1 AND R_TRIG_1.Q THEN CARTONNO1:=CARTONNO_DIS;
ELSIF PRGNO_LOAD=4 AND R_TRIG_1.Q THEN CARTONNO4:=CARTONNO_DIS;
ELSIF PRGNO_LOAD=5 AND R_TRIG_1.Q THEN CARTONNO5:=CARTONNO_DIS;
ELSIF PRGNO_LOAD=6 AND R_TRIG_1.Q THEN CARTONNO6:=CARTONNO_DIS;
ELSIF PRGNO_LOAD=7 AND R_TRIG_1.Q THEN CARTONNO7:=CARTONNO_DIS;
ELSIF PRGNO_LOAD=8 AND R_TRIG_1.Q THEN CARTONNO8:=CARTONNO_DIS;
ELSIF PRGNO_LOAD=9 AND R_TRIG_1.Q THEN CARTONNO9:=CARTONNO_DIS;
ELSIF PRGNO_LOAD=10 AND R_TRIG_1.Q THEN CARTONNO10:=CARTONNO_DIS;
END_IF

DefaultNetWt :=DFLTNETWT_DIS;
NetWtTolRep:=	NETWTTOL_DIS;
DefaultGrossWt:=	DFLTGROSSWT_DIS;
GrossWtTolRep:=	GROSSWTTOL_DIS;
END_PROGRAM

(* POU AutoMode/DATALOG_PRINT, ST *)
PROGRAM DATALOG_PRINT
VAR
	step: INT;
	bOpen: BOOL;
	FB_FileOpen1: FB_FileOpen;
	(*sPrintPath: STRING(80):= '\\PLC-PC\Reports\Print.csv';*)
	FB_FileWrite1: FB_FileWrite;
	FB_FileClose1: FB_FileClose;
	FB_FileDelete1: FB_FileDelete;

	TON_1: TON;
	bOpen1: BOOL;
	sHeadline: STRING;
	sData: STRING;
	ProductionData_PrintData: ProductionData_PrintData;
	PrintEnabled: BOOL;

	Timer_1: TON;
	Timer_2: TON;
	TON_2: TON;
	BlendPrint: STRING;
	WriteError: INT;
	TON_writedly: TON;
	OpenError: INT;
	TON_Opendly: TON;

END_VAR
IF PrintEnableHmi THEN PrintEnabled:=TRUE;PrintValue:=1;ELSE PrintEnabled:=FALSE;PrintValue:=0;END_IF


BlendPrint:=CONCAT(BLEND_DIS, '%');


		(*ProductionData_PrintData.Print						:=INT_TO_STRING( PrintValue );
		ProductionData_PrintData.ConeType1				:=(COUNT_DIS);
		ProductionData_PrintData.Blend1					:=(BLEND_DIS);
		ProductionData_PrintData.DefaultnetWt1				:=(NetwtPrint);
		ProductionData_PrintData.DefaultGrossWt1			:=(GrosswtPrint);
		ProductionData_PrintData.LotNo1					:=(LOTNO_DIS);
		ProductionData_PrintData.BagNo1					:=DINT_TO_STRING(CARTONNO_DIS);
		ProductionData_PrintData.ConeTip1					:=(CONETIP_DIS);
		ProductionData_PrintData.Shade1					:=(SHADE_DIS);
		ProductionData_PrintData.PackType1					:=(PACKTYPE_DIS);
		ProductionData_PrintData.Cones1					:=DINT_TO_STRING(iATotalNoOfCones);*)


ProductionData_PrintData.Print						:=INT_TO_STRING( PrintValue );
ProductionData_PrintData.PgNo						:=DINT_TO_STRING( PRGNO_DIS );
ProductionData_PrintData.TotNoCones						:=INT_TO_STRING( iATotalNoOfCones );
ProductionData_PrintData.CartNo						:=DINT_TO_STRING(CARTONNO_DIS);
ProductionData_PrintData.LotNo						:=(LOTNO_DIS);
ProductionData_PrintData.DateTi						:=(sDATEFinal);
ProductionData_PrintData.NetWt						:=REAL_TO_STRING(DFLTNETWT_DIS);
ProductionData_PrintData.WrkOrdNo						:=(WORKORDERNO_DIS);
ProductionData_PrintData.DfltNetWt						:=REAL_TO_STRING(* (DFLTNETWT_DIS);*)(EmptyConeWtRep);
ProductionData_PrintData.DfltGrsWt						:=REAL_TO_STRING(DFLTGROSSWT_DIS);
ProductionData_PrintData.Blnd						:=(BlendPrint);
ProductionData_PrintData.Shd						:=(SHADE_DIS );
ProductionData_PrintData.ConeTip						:=(CONETIP_DIS);
ProductionData_PrintData.ConeNetWt						:=REAL_TO_STRING(CONENETWT_DIS);
ProductionData_PrintData.ConeLenght						:=REAL_TO_STRING (CONELENGTH_DIS);
ProductionData_PrintData.Dom						:=(DOM_EXPORT_DIS);
ProductionData_PrintData.Pack						:=(PACKTYPE_DIS);
ProductionData_PrintData.CountCod						:=(COUNT_DIS);


	(*	(*	######## LOG PRODUCTION DATA		#####	*)

ProductionDataValues_Print:= CONCAT(ProductionData_PrintData.Print,',');
ProductionDataValues_Print:=	 CONCAT( ProductionDataValues_Print,ProductionData_PrintData.ConeType1);
ProductionDataValues_Print:= CONCAT( ProductionDataValues_Print,',');
ProductionDataValues_Print:=	 CONCAT( ProductionDataValues_Print,ProductionData_PrintData.Blend1);
ProductionDataValues_Print:= CONCAT( ProductionDataValues_Print,',');
ProductionDataValues_Print:=	 CONCAT( ProductionDataValues_Print,ProductionData_PrintData.DefaultnetWt1);
ProductionDataValues_Print:= CONCAT( ProductionDataValues_Print,',');
ProductionDataValues_Print:=	 CONCAT( ProductionDataValues_Print,ProductionData_PrintData.DefaultGrossWt1);
ProductionDataValues_Print:= CONCAT( ProductionDataValues_Print,',');
ProductionDataValues_Print:=	 CONCAT( ProductionDataValues_Print,ProductionData_PrintData.LotNo1);
ProductionDataValues_Print:= CONCAT( ProductionDataValues_Print,',');
ProductionDataValues_Print:=	 CONCAT( ProductionDataValues_Print,ProductionData_PrintData.BagNo1);
ProductionDataValues_Print:= CONCAT( ProductionDataValues_Print,',');
ProductionDataValues_Print:=	 CONCAT( ProductionDataValues_Print,ProductionData_PrintData.ConeTip1);
ProductionDataValues_Print:= CONCAT( ProductionDataValues_Print,',');
ProductionDataValues_Print:=	 CONCAT( ProductionDataValues_Print,ProductionData_PrintData.PackType1);
ProductionDataValues_Print:= CONCAT( ProductionDataValues_Print,',');
ProductionDataValues_Print:=	 CONCAT( ProductionDataValues_Print,ProductionData_PrintData.Cones1);
ProductionDataValues_Print:= CONCAT( ProductionDataValues_Print,',');
ProductionDataValues_Print:=	 CONCAT( ProductionDataValues_Print,ProductionData_PrintData.Shade1);
ProductionDataValues_Print:= CONCAT( ProductionDataValues_Print,'$0A');*)
	(*	######## LOG PRODUCTION DATA		#####	*)

ProductionDataValues_Print:= CONCAT(ProductionData_PrintData.Print,',');
ProductionDataValues_Print:=	 CONCAT( ProductionDataValues_Print,ProductionData_PrintData.CountCod);
ProductionDataValues_Print:= CONCAT( ProductionDataValues_Print,',');
ProductionDataValues_Print:=	 CONCAT( ProductionDataValues_Print,ProductionData_PrintData.Blnd);
ProductionDataValues_Print:= CONCAT( ProductionDataValues_Print,',');
ProductionDataValues_Print:=	 CONCAT( ProductionDataValues_Print,ProductionData_PrintData.NetWt);
ProductionDataValues_Print:= CONCAT( ProductionDataValues_Print,',');
ProductionDataValues_Print:=	 CONCAT( ProductionDataValues_Print,ProductionData_PrintData.DfltGrsWt);
ProductionDataValues_Print:= CONCAT( ProductionDataValues_Print,',');
ProductionDataValues_Print:=	 CONCAT( ProductionDataValues_Print,ProductionData_PrintData.LotNo);
ProductionDataValues_Print:= CONCAT( ProductionDataValues_Print,',');
ProductionDataValues_Print:=	 CONCAT( ProductionDataValues_Print,ProductionData_PrintData.CartNo);
ProductionDataValues_Print:= CONCAT( ProductionDataValues_Print,',');
ProductionDataValues_Print:=	 CONCAT( ProductionDataValues_Print,ProductionData_PrintData.ConeTip);
ProductionDataValues_Print:= CONCAT( ProductionDataValues_Print,',');
ProductionDataValues_Print:=	 CONCAT( ProductionDataValues_Print,ProductionData_PrintData.Pack);
ProductionDataValues_Print:= CONCAT( ProductionDataValues_Print,',');
ProductionDataValues_Print:=	 CONCAT( ProductionDataValues_Print,ProductionData_PrintData.TotNoCones);
ProductionDataValues_Print:= CONCAT( ProductionDataValues_Print,',');
ProductionDataValues_Print:=	 CONCAT( ProductionDataValues_Print,ProductionData_PrintData.Shd);
ProductionDataValues_Print:= CONCAT( ProductionDataValues_Print,',');
ProductionDataValues_Print:=	 CONCAT( ProductionDataValues_Print,ProductionData_PrintData.ConeNetWt);
ProductionDataValues_Print:= CONCAT( ProductionDataValues_Print,',');
ProductionDataValues_Print:=	 CONCAT( ProductionDataValues_Print,ProductionData_PrintData.ConeLenght);
ProductionDataValues_Print:= CONCAT( ProductionDataValues_Print,'$0A');
(*ProductionDataValues_Print:=	 CONCAT( ProductionDataValues_Print,ProductionData_PrintData.WrkOrdNo);
ProductionDataValues_Print:= CONCAT( ProductionDataValues_Print,',');
ProductionDataValues_Print:=	 CONCAT( ProductionDataValues_Print,ProductionData_PrintData.DfltNetWt);
ProductionDataValues_Print:= CONCAT( ProductionDataValues_Print,',');
ProductionDataValues_Print:=	 CONCAT( ProductionDataValues_Print,ProductionData_PrintData.Dom);
ProductionDataValues_Print:= CONCAT( ProductionDataValues_Print,'$0A');*)




(*
ProductionData_Print:= CONCAT( 'Print',',');
		ProductionData_Print:=	 CONCAT( ProductionData_Print,'Count Type');
		ProductionData_Print:= CONCAT( ProductionData_Print,',');
ProductionData_Print:=	 CONCAT( ProductionData_Print,'Blend');
		ProductionData_Print:= CONCAT( ProductionData_Print,',');
ProductionData_Print:=	 CONCAT( ProductionData_Print,'NetWt');
		ProductionData_Print:= CONCAT( ProductionData_Print,',');
ProductionData_Print:=	 CONCAT( ProductionData_Print,'Grss Wt');
		ProductionData_Print:= CONCAT( ProductionData_Print,',');
ProductionData_Print:=	 CONCAT( ProductionData_Print,'Lot No');
		ProductionData_Print:= CONCAT( ProductionData_Print,',');
ProductionData_Print:=	 CONCAT( ProductionData_Print,'Bag No');
		ProductionData_Print:= CONCAT( ProductionData_Print,',');
ProductionData_Print:=	 CONCAT( ProductionData_Print,'Cone Tip');
		ProductionData_Print:= CONCAT( ProductionData_Print,',');
ProductionData_Print:=	 CONCAT( ProductionData_Print,'PackType1');
		ProductionData_Print:= CONCAT( ProductionData_Print,',');
ProductionData_Print:=	 CONCAT( ProductionData_Print,'Cones');
		ProductionData_Print:= CONCAT( ProductionData_Print,',');
ProductionData_Print:=	 CONCAT( ProductionData_Print,'Shade');
		ProductionData_Print:= CONCAT( ProductionData_Print,'$0A');*)



ProductionData_Print:= CONCAT( 'Print',',');
	ProductionData_Print:=	 CONCAT( ProductionData_Print,'Count');
ProductionData_Print:= CONCAT( ProductionData_Print,',');
	ProductionData_Print:=	 CONCAT( ProductionData_Print,'Blend');
ProductionData_Print:= CONCAT( ProductionData_Print,',');
	ProductionData_Print:=	 CONCAT( ProductionData_Print,'NetWt');
ProductionData_Print:= CONCAT( ProductionData_Print,',');
         ProductionData_Print:=	 CONCAT( ProductionData_Print,'GrossWt');
ProductionData_Print:= CONCAT( ProductionData_Print,',');
	ProductionData_Print:=	 CONCAT( ProductionData_Print,'LotNo');
ProductionData_Print:= CONCAT( ProductionData_Print,',');

	ProductionData_Print:=	 CONCAT( ProductionData_Print,'CartonNo');
ProductionData_Print:= CONCAT( ProductionData_Print,',');
	ProductionData_Print:=	 CONCAT( ProductionData_Print,'ConeTip');
ProductionData_Print:= CONCAT( ProductionData_Print,',');
	ProductionData_Print:=	 CONCAT( ProductionData_Print,'Pack');
ProductionData_Print:= CONCAT( ProductionData_Print,',');
	ProductionData_Print:=	 CONCAT( ProductionData_Print,'TotNoCone');
ProductionData_Print:= CONCAT( ProductionData_Print,',');

	ProductionData_Print:=	 CONCAT( ProductionData_Print,'Shade');
ProductionData_Print:= CONCAT( ProductionData_Print,',');
	ProductionData_Print:=	 CONCAT( ProductionData_Print,'ConeNetWt');
ProductionData_Print:= CONCAT( ProductionData_Print,',');

ProductionData_Print:=	 CONCAT( ProductionData_Print,'ConeLeng');
		ProductionData_Print:= CONCAT( ProductionData_Print,'$0A');
(*ProductionData_Print:=	 CONCAT( ProductionData_Print,'WorkOrdNo');
		ProductionData_Print:= CONCAT( ProductionData_Print,',');
ProductionData_Print:=	 CONCAT( ProductionData_Print,'DfltNtWt');
		ProductionData_Print:= CONCAT( ProductionData_Print,',');
ProductionData_Print:=	 CONCAT( ProductionData_Print,'Dom');
		ProductionData_Print:= CONCAT( ProductionData_Print,'$0A');*)





FB_FileOpen1(
	sNetId:='192.168.225.201.1.1',
	sPathName:= '\\ACP\Reports\productiondata.csv' ,
	nMode:=FOPEN_MODEAPPEND ,
	ePath:=PATH_GENERIC ,
	bExecute:= ,
	tTimeout:=T#2s ,
	bBusy=> ,
	bError=> ,
	nErrId=> ,
	hFile=> );

FB_FileWrite1(
	sNetId:='192.168.225.201.1.1',
	hFile:=FB_FileOpen1.hFile ,
	pWriteBuff:=ADR(ProductionDataValues_Print_Com),
	cbWriteLen:=LEN(ProductionDataValues_Print_Com),
	bExecute:= ,
	tTimeout:=T#2s ,
	bBusy=> ,
	bError=> ,
	nErrId=> ,
	cbWrite=> );


FB_FileClose1(
	sNetId:='192.168.225.201.1.1',
	hFile:=FB_FileOpen1.hFile ,
	bExecute:= ,
	tTimeout:=T#2s ,
	bBusy=> ,
	bError=> ,
	nErrId=> );

FB_FileDelete1(
	sNetId:='192.168.225.201.1.1' ,
	sPathName:= '\\ACP\Reports\productiondata.csv' ,
	ePath:=PATH_GENERIC ,
	bExecute:= ,
	tTimeout:=T#2s ,
	bBusy=> ,
	bError=> ,
	nErrId=> );

CASE step OF

0: IF PrintOk THEN
	TON_2(IN:=FALSE);

	FB_FileOpen1.bExecute:=TRUE;
	IF NOT FB_FileOpen1.bBusy AND NOT FB_FileOpen1.bError AND FB_FileOpen1.hFile>0 THEN bOpen1:=FALSE; step:=step+1;END_IF
	END_IF


1:	IF NOT FB_FileOpen1.bBusy AND NOT FB_FileOpen1.bError AND FB_FileOpen1.hFile>0 THEN bOpen1:=FALSE; PrintOk:=FALSE;step:=step+1;END_IF

2:
	ProductionDataValues_Print_Com:=ProductionData_Print;
	FB_FileWrite1.bExecute:=TRUE;
	IF NOT FB_FileWrite1.bBusy AND NOT FB_FileWrite1.bError THEN step:=step+1;END_IF


3:	IF NOT FB_FileWrite1.bBusy AND NOT FB_FileWrite1.bError THEN FB_FileWrite1.bExecute:=FALSE; step:=step+1;END_IF

4:	ProductionDataValues_Print_Com:=ProductionDataValues_Print;
	FB_FileWrite1.bExecute:=TRUE;
	IF NOT FB_FileWrite1.bBusy AND NOT FB_FileWrite1.bError THEN step:=step+1;END_IF



5:	step:=step+1;


6:	IF NOT FB_FileWrite1.bBusy AND NOT FB_FileWrite1.bError THEN FB_FileWrite1.bExecute:=FALSE; step:=step+1;END_IF


7:	FB_FileClose1.bExecute:=TRUE;
	 IF NOT FB_FileClose1.bBusy AND NOT FB_FileClose1.bError THEN  step:=step+1;END_IF

8:	TON_1(IN:=TRUE , PT:=t#1s , Q=> , ET=> );
	IF TON_1.Q THEN step:=step+1;END_IF

9:	IF NOT FB_FileDelete1.bBusy AND NOT FB_FileDelete1.bError THEN
	TON_1(IN:=FALSE);
	(*FB_FileDelete1.bExecute:=TRUE;*)step:=step+1;END_IF

10:
	FB_FileOpen1.bExecute:=FALSE;
	FB_FileWrite1.bExecute:=FALSE;
	FB_FileClose1.bExecute:=FALSE;
	FB_FileDelete1.bExecute:=FALSE;
	bOpen:=FALSE;step:=step+1;

11:		TON_2(IN:=TRUE , PT:=t#10s , Q=> , ET=> );
	IF TON_2.Q THEN(* PrintOk:=TRUE;	*) step:=0;END_IF

END_CASE



CASE WriteError OF

0:	IF FB_FileWrite1.bError THEN FB_FileWrite1.bExecute:=FALSE;TON_writedly(IN:=FALSE);
	WriteError:=WriteError+1;END_IF

1:	TON_writedly(IN:=TRUE , PT:=t#2s , Q=> , ET=> );
	IF TON_writedly.Q THEN FB_FileWrite1.bExecute:=TRUE;WriteError:=WriteError+1;END_IF

2:	TON_writedly(IN:=FALSE);WriteError:=0;

END_CASE




CASE OpenError OF

0:	IF FB_FileOpen1.bError THEN FB_FileOpen1.bExecute:=FALSE;TON_Opendly(IN:=FALSE);
	OpenError:=OpenError+1;END_IF

1:	TON_Opendly(IN:=TRUE , PT:=t#2s , Q=> , ET=> );
	IF TON_Opendly.Q THEN FB_FileOpen1.bExecute:=TRUE;OpenError:=OpenError+1;END_IF

2:	TON_Opendly(IN:=FALSE);OpenError:=0;

END_CASE
END_PROGRAM

(* POU AutoMode/One_Min_Conv, ST *)
PROGRAM One_Min_Conv
VAR
	TON_5: TON;
	TON_6: TON;
	rGrossWtTolMin: REAL;
	rGrossWtTolMax: REAL;
	bGrossWieghtOkTemp: BOOL;
	bQAGrossWtPiston1: BOOL;
	bcheck: BOOL;

	TEST1: BOOL;
	TEST2: BOOL;
	tGrossWtEndSenDly: TON;
	CylErrChkBit: BOOL;
END_VAR
IF NOT  bIEmergency   OR bStopHmi  OR  bAutoModeOff  OR bIMCStop THEN
One_Min_Conv_1:=0;
bQGross_Roller_On:=FALSE; TON_5(IN:=FALSE); TON_6(IN:=FALSE);
END_IF
rGrossWtTolMax:= (DFLTGROSSWT_DIS + GROSSWTTOL_DIS);

rGrossWtTolMin:= (DFLTGROSSWT_DIS - GROSSWTTOL_DIS);


CASE One_Min_Conv_1 OF


	0:	IF bAutoModeOn AND bIGross_Crossing_Input  AND bAMcStartInAuto   AND NOT bAPauseSeq THEN
		bQGross_Roller_On:=TRUE; TON_5(IN:=FALSE);
		One_Min_Conv_1:=One_Min_Conv_1+1; END_IF

	1:	TON_5(IN:=TRUE , PT:=t#10S , Q=> , ET=> );
		IF  bIGross_Weight_Stop   AND NOT bAPauseSeq AND NOT  TON_5.Q THEN  One_Min_Conv_1:=One_Min_Conv_1+1;
		ELSE
		 IF  TON_5.Q THEN bcheck:=TRUE;  bQGross_Roller_On:=FALSE;  One_Min_Conv_1:=0;
		END_IF
		END_IF

	2:	IF bAutoModeOn AND bIGross_Weight_Stop   AND NOT bAPauseSeq THEN
		tGrossWtEndSenDly(IN:= FALSE);
		bQGross_Roller_On:=FALSE; bQGross_Cylinder_On:=TRUE;
		(*tGrossWtEndSenDly(IN:= TRUE, PT:=t#5s , Q=> , ET=> ); *)
		CylErrChkBit:=TRUE;
		One_Min_Conv_1:=One_Min_Conv_1+1; END_IF

	3:	IF bIGross_Cyl_End THEN 	CylErrChkBit:=FALSE; One_Min_Conv_1:=One_Min_Conv_1+1;
		ELSIF NOT bIGross_Cyl_End AND tGrossWtEndSenDly.Q THEN
		bGrossWtCylEndSenError:=TRUE;
		SGrossWtCylEndSenErrMsg:='Gross weight Cyl End Sensor Error';
		One_Min_Conv_1:=13;
		END_IF

	4:	TON_6(IN:=TRUE , PT:=t#9.5S , Q=> , ET=> );
		 IF  TON_6.Q THEN One_Min_Conv_1:=One_Min_Conv_1+1;  END_IF

	5:	IF  rGrossWeight >=rGrossWtTolMin  AND  rGrossWeight  <= rGrossWtTolMax  THEN
		bGrossWieghtOkTemp:=TRUE; rGrossWeighToReport:=rGrossWeight ;  bGrossWieghtNokTemp:=FALSE;
		One_Min_Conv_1:=One_Min_Conv_1+1;
		ELSIF  rGrossWeight  >  rGrossWtTolMax THEN
		bGrossWieghtNokTemp:=TRUE; bGrossWieghtOkTemp:=FALSE;
		One_Min_Conv_1:=One_Min_Conv_1+2;
		ELSIF   rGrossWeight  < rGrossWtTolMin   THEN
		bGrossWieghtNokTemp:=TRUE; bGrossWieghtOkTemp:=FALSE;
		One_Min_Conv_1:=One_Min_Conv_1+2;
		END_IF

	6:	IF bGrossWieghtOkTemp (*AND TEST1*)  THEN bGrossWieghtOk:=TRUE; bQAGrossWieghtOkIndi:=TRUE; One_Min_Conv_1:=One_Min_Conv_1+2;  TON_6(IN:=FALSE);  END_IF

	7:	IF bGrossWieghtNokTemp  (*AND TEST2 *)THEN bGrossWieghtNOk:=TRUE;
		SGrossWtNokMsg:='Gross Weight is Less OR more';
		bReadGWieght:=FALSE; One_Min_Conv_1:=One_Min_Conv_1+2;   TON_6(IN:=FALSE); END_IF


	8:	IF bGrossWieghtOk (*  AND NOT bGrossWieghtNok *) AND bAutoModeOn  AND NOT bAPauseSeq THEN
		 bQGross_Cylinder_On:=FALSE; bReadGWieght:=FALSE; bGrossWieghtOkTemp:=FALSE;
		bQAGrossWieghtOkIndi:=FALSE;   (*====== Modified for  Gross  Weight   bypass  ==============*)
		bACyclePass:=TRUE;
		GrossWtReedSwBit:=TRUE;
		One_Min_Conv_1:=One_Min_Conv_1+2;
		 END_IF

	9:	IF bErrorReset THEN  bGrossWieghtNOk:=FALSE;
		SGrossWtNokMsg:='';
		One_Min_Conv_1:=4; END_IF

	10:	IF bIGross_Cyl_Home  AND NOT bAGrossWtHomeSenRsError THEN GrossWtReedSwBit:=FALSE ; bQGross_Roller_On:=TRUE;  One_Min_Conv_1:=One_Min_Conv_1+1;END_IF

	11:	bACyclePass:=FALSE;One_Min_Conv_1:=One_Min_Conv_1+1;

	12:	IF bAutoModeOn AND NOT  bIGross_Weight_Stop   AND NOT bAPauseSeq THEN
		 One_Min_Conv_1:=0;  bQGross_Roller_On:=FALSE; END_IF

	13:	IF bErrorReset AND bIGross_Cyl_End THEN
		CylErrChkBit:=FALSE;
		bGrossWtCylEndSenError:=FALSE;
		tGrossWtEndSenDly(IN:= FALSE);
		SGrossWtCylEndSenErrMsg:='';
		One_Min_Conv_1:=2;
		ELSIF NOT bIGross_Cyl_End AND bErrorReset THEN
		CylErrChkBit:=FALSE;
		bGrossWtCylEndSenError:=FALSE;
		tGrossWtEndSenDly(IN:= FALSE);
		SGrossWtCylEndSenErrMsg:='';
		One_Min_Conv_1:=2;
		END_IF
END_CASE





IF CylErrChkBit THEN tGrossWtEndSenDly(IN:= TRUE, PT:=t#5s , Q=> , ET=> );
END_IF
END_PROGRAM

(* POU AutoMode/FlimRollerUnit, ST *)
PROGRAM FlimRollerUnit
VAR
	step: INT;
	bQAFilmRollerMotor1OnAuto: BOOL;
	bQAFilmRollerMotor2OnAuto: BOOL;
	bQAFilmRollerMotor3OnAuto: BOOL;
END_VAR
bQAFilmRollerMotor1:= ( bQAFilmRollerMotor1OnAuto );

bQAFilmRollerMotor2:= ( bQAFilmRollerMotor2OnAuto );

bQAFilmRollerMotor3:=( bQAFilmRollerMotor3OnAuto );





		IF NOT 	bIWrappingFilmTensionPlate_1  THEN
		bQAFilmRollerMotor1OnAuto:=TRUE;
		ELSE
		bQAFilmRollerMotor1OnAuto:=FALSE;
		END_IF


		IF NOT	bIWrappingFilmTensionPlate_2   THEN
		bQAFilmRollerMotor2OnAuto:=TRUE;
		ELSE
		bQAFilmRollerMotor2OnAuto:=FALSE;
		END_IF



		IF NOT	bIWrappingFilmTensionPlate_3    THEN
		bQAFilmRollerMotor3OnAuto:=TRUE;
		ELSE
		bQAFilmRollerMotor3OnAuto:=FALSE;
		END_IF
END_PROGRAM

(* POU AutoMode/Auto, ST *)
PROGRAM Auto
VAR
	Timer1: TON;
	Timer2: TON;
	bAmber: BOOL;
	bAGreen: BOOL;
	bARed: BOOL;
	bABuzzertest: BOOL;
	bABuzzertemp: BOOL;
	bAmberTemp: BOOL;
	bAmberbit1: BOOL;
END_VAR
	IF bAutoModeOn AND bIMCStart THEN bAMcStartInAuto:=TRUE; bAStop:=FALSE;  END_IF

	IF NOT bIEmergency OR  bIMCStop OR bStopHmi   THEN bAMcStartInAuto:=FALSE; END_IF


IF bAutoModeOff THEN bAMcStartInAuto:=FALSE; END_IF




(*=================Model Selection Logic===============*)

IF b12ConeModelHmi AND NOT  b18ConeModelHmi AND NOT  b24ConeModelHmi AND NOT b32ConeModelHmi AND NOT bInterlockInitial_2 THEN
b12ConeModelSelected:=TRUE; b16ConeModelSelected:=FALSE; b18ConeModelSelected:=FALSE; b24ConeModelSelected:=FALSE; b32ConeModelSelected:=FALSE;  END_IF

IF NOT  b12ConeModelHmi AND   b18ConeModelHmi AND NOT  b24ConeModelHmi AND NOT b32ConeModelHmi AND NOT bInterlockInitial_2 THEN
b18ConeModelSelected:=TRUE;   b16ConeModelSelected:=FALSE; b12ConeModelSelected:=FALSE; b24ConeModelSelected:=FALSE; b32ConeModelSelected:=FALSE;   END_IF

IF  NOT b12ConeModelHmi AND NOT  b18ConeModelHmi AND   b24ConeModelHmi AND NOT b32ConeModelHmi AND NOT bInterlockInitial_2 THEN
 b24ConeModelSelected:=TRUE; b16ConeModelSelected:=FALSE;  b18ConeModelSelected:=FALSE; b12ConeModelSelected:=FALSE; b32ConeModelSelected:=FALSE;    END_IF

IF  NOT b12ConeModelHmi AND NOT  b18ConeModelHmi AND NOT  b24ConeModelHmi AND  b32ConeModelHmi AND NOT bInterlockInitial_2  THEN
b32ConeModelSelected:=TRUE;  b18ConeModelSelected:=FALSE; b24ConeModelSelected:=FALSE; b12ConeModelSelected:=FALSE;    END_IF

IF  b16ConeModelHmi AND NOT b12ConeModelHmi AND NOT  b18ConeModelHmi AND NOT  b24ConeModelHmi AND  NOT b32ConeModelHmi  AND NOT bInterlockInitial_2 THEN
 b16ConeModelSelected:=TRUE;b32ConeModelSelected:=FALSE;  b18ConeModelSelected:=FALSE; b24ConeModelSelected:=FALSE; b12ConeModelSelected:=FALSE;    END_IF


IF b12ConeModelSelected THEN iATotalNoOfCones:=12;
ELSIF b16ConeModelSelected THEN iATotalNoOfCones:=16;
ELSIF  b18ConeModelSelected THEN iATotalNoOfCones:=18;
ELSIF  b24ConeModelSelected THEN iATotalNoOfCones:=24;
ELSIF  b32ConeModelSelected THEN iATotalNoOfCones:=32;
END_IF


Timer1(IN:=(bAInializeStarted AND NOT Timer2.Q   ) ,  PT:=t#0.5s , Q=> , ET=>, );
Timer2(IN:= Timer1.Q, PT:=t#0.5s , Q=> , ET=> );

IF bIMCStart THEN bAGreen:=TRUE; END_IF

IF Timer1.Q    AND NOT  bAError   AND NOT bAStop AND NOT bAPauseSeq THEN bAmber :=TRUE; bAGreen:=FALSE;  ELSE  bAmber:=FALSE; END_IF

IF Timer1.Q OR bAMcRunninig   OR bAMcReady AND NOT bAError AND NOT bAStop  THEN bAGreen :=TRUE;   ELSE  bAGreen:=FALSE; END_IF

IF Timer1.Q OR bAStop OR  bStopHmi THEN bARed :=TRUE; (*bAGreen:=FALSE;*)  bABuzzer:=FALSE; ELSE  bARed:=FALSE; END_IF
IF  bAPauseSeq THEN bAmberbit1 :=TRUE; bAGreen:=FALSE; ELSE bAmberbit1 :=FALSE; END_IF
IF Timer1.Q  AND NOT bAPauseSeq THEN  bAmber :=TRUE;  ELSE  bAmber :=FALSE;END_IF
IF bAError THEN  bAmberbit2:=TRUE;bAGreen:=FALSE;ELSE bAmberbit2 :=FALSE;END_IF

bQAAmber:=bAmber  OR bABuzzer OR bAmberbit1 OR bAmberbit2 ;
bQAGreen:= bAGreen;
bQARed:=bARed;
 bQABuzzer:= bABuzzer;

IF NOT  bIEmergency OR bStopHmi  OR bAutoModeOff OR bIMCStop  THEN bARed :=TRUE; bAGreen:=FALSE; bAmber:=FALSE; bAMcRunninig:=FALSE; END_IF
END_PROGRAM

(* POU AutoMode/UnitA_RowStopper, ST *)
PROGRAM UnitA_RowStopper
VAR
	step: INT;

	iSensorOnVal:UINT;
	CTU_1Enable: BOOL;
	R_TRIG_1: F_TRIG;
	CTU_2: CTU;
	R_TRIG_2: R_TRIG;
	tRowStopperRevDly1: TON;
	UnitAConeCrossCount: CTU;
	test: BOOL;
	bStopRetUnitA: BOOL;
	RowStopperMotorStopDly: TON;
	bRetUnitAStarttemp: BOOL;
	bAUnitAWeighOktemp: BOOL;
	RowStopperEndRSErrorDly: TON;
	bStartTemp1: BOOL;
	UnitAOverTemp: BOOL;
	RowStopperEndSenErr: BOOL;
	interLockStep: INT;
	UnitACompleteCheckCountCv: INT;
	bEnableBit1: BOOL;
	UnitAConeCross: CTU;
	Testtimer: TON;
	bAUnitBConeCrossingOff_2: BOOL;
	step3: INT;
	TON_7: TON;
	R_TRIG_4: R_TRIG;
	timer3: TON;

	SenSelect_1: SenSelect;
	iAConeCrossCount: INT;
	bQAUnitA_RowStopperMotorFwd2: BOOL;
	bQAUnitA_RowStopperMotorFwd1: BOOL;
	bQAUnitA_RowStopperMotorRev1: BOOL;
	sRetreivalAStatus: STRING;
	bRetUnitARst: BOOL;
	iAConeCrossCounttemp: INT;
	GetDLy: TON;
	bCheckSensor: BOOL;
	tConeChkDly: TON;
	bUnitAConeMiss:BOOL ;
	iAConeCrossPVal: INT;
	tConeCrossDly: TON;
	step2: INT;
	F_TRIG_5: F_TRIG;
	TON_6: TON;
	bAUnitBConeCrossing_1: BOOL;
	bAUnitBConeCrossingOff: BOOL;
	step4: INT;
	TON_8: TON;
	bAUnitAConeCrossing_1: BOOL;
	TON_9: TON;
	bAUnitAConeCrossingOff: BOOL;
	TON_10: TON;
	F_TRIG_3: F_TRIG;
	CountAtLimitBNok: BOOL;
	CountCheckdly: TON;
	UnitAConeCompChkCount: CTU;
	tRowStopperMidDly1: TON;
	tUnitACountDelay1: TON;
	TEnableCounter: BOOL;
	CompleteTestbitA: BOOL;
	bCounterLockUnitA: BOOL;
	bStartUnitaCompCount: BOOL;
END_VAR
UnitASenSelet:=iSensorOnVal;

(*=============Checking the No of sensors sensed================*)

IF bCheckSensor THEN
SenSelect_1(
		bVarIn1:=bIUnitAConeDetection1 ,
		bVarIn2:= bIUnitAConeDetection2,
		bVarIn3:= bIUnitAConeDetection3,
		bVarIn4:= bIUnitAConeDetection4,
		ByteResult=>iSensorOnVal );


END_IF

IF iSensorOnVal=15 THEN iAConeCrossCount:=4;
		ELSIF  iSensorOnVal=14 THEN iAConeCrossCount:=3;
		ELSIF  iSensorOnVal=13 THEN iAConeCrossCount:=3;
		ELSIF  iSensorOnVal=12 THEN iAConeCrossCount:=2;
		ELSIF  iSensorOnVal=11 THEN iAConeCrossCount:=3;
		ELSIF  iSensorOnVal=10 THEN iAConeCrossCount:=2;
		ELSIF  iSensorOnVal=9 THEN iAConeCrossCount:=2;
		ELSIF  iSensorOnVal=8 THEN iAConeCrossCount:=1;
		ELSIF  iSensorOnVal=7 THEN iAConeCrossCount:=3;
		ELSIF  iSensorOnVal=6 THEN iAConeCrossCount:=2;
		ELSIF  iSensorOnVal=5 THEN iAConeCrossCount:=2;
		ELSIF  iSensorOnVal=4 THEN iAConeCrossCount:=1;
		ELSIF  iSensorOnVal=3 THEN iAConeCrossCount:=2;
		ELSIF  iSensorOnVal=2 THEN iAConeCrossCount:=1;
		ELSIF  iSensorOnVal=1 THEN iAConeCrossCount:=1;
		END_IF





bQAUnitA_RowStopperMotorForward1:=( bQAUnitA_RowStopperMotorFwd1 OR bQAUnitA_RowStopperMotorFwd2 );

bQAUnitA_RowStopperMotorReverse1:= ( bQAUnitA_RowStopperMotorRev1 OR bRetUnitARst );

CASE step OF

	0:	IF bAutoModeOn AND bAUnitAWeighOk  AND bRetUnitAStart   AND NOT bAInializeStarted  AND NOT bIntialAckBit  AND bInterlockInitial_2 THEN
		CTU_2.RESET:=TRUE;

		step:=step+1;
		END_IF

	1:	PROCESSCOMPLETE:=FALSE;step:=step+1;

	2:	IF bAutoModeOn(* AND bIUnitA_LiftPistonHome  *)THEN
		step:=step+1;


		END_IF

	3:	UnitAConeCompChkCount.RESET:=FALSE;
		TestTimer(IN:=FALSE);
		step:=step+1;

	4:	IF bAutoModeOn    AND NOT bUnitBRowStopperStarted  AND NOT ConeInCompleteB  (*ConeInCompleteTestbitB*)
		AND NOT bAPauseSeq  AND NOT ConeInCompleteA   AND bInterlockInitial_2 THEN
		bQAUnitA_RowStopperMotorFwd1:=TRUE;
		UnitAConeCrossCount.RESET:=TRUE;
		bAUnitAWeighOk:=FALSE;

		bUnitARowStopperStarted:=TRUE;
		sRetreivalAStatus:= 'Running';

		 step:=step+1;
		END_IF

	5:	RowStopperMotorStopDly(In:=FALSE);
		 step:=step+1;

	6:	IF bIUnitAConeDetection1 OR  bIUnitAConeDetection2 OR  bIUnitAConeDetection3 OR   bIUnitAConeDetection4  THEN

		step:=step+1;
		ELSIF NOT bIUnitAConedetection1 AND NOT  bIUnitAConedetection2 AND NOT  bIUnitAConedetection3 AND NOT bIUnitAConeDetection4 AND  bIUnitA_RowStopperEnd THEN

		step:=15;
		END_IF

	7:	CompleteTestbitA:=FALSE;
		RowStopperMotorStopDly( IN:=TRUE , PT:=T#0.4s , Q=> , ET=> );
		IF RowStopperMotorStopDly.Q THEN  UnitAConeCrossCount.RESET:=FALSE;  step:=step+1; END_IF


	8:	bStartUnitaCompCount:=TRUE;
		bQAUnitA_RowStopperMotorFwd1:=FALSE;
		GetDLy(IN:=FALSE);
		tRowStopperRevDly1(IN:=FALSE);
		step:=step+1;

	9:	 IF  NOT   bAPauseSeq THEN  bCheckSensor:=TRUE;

		step:=step+1;

		END_IF


	10:	GetDLy(IN:=TRUE , PT:=t#0.4s , Q=> , ET=> );
		 IF GetDLy.Q THEN bCheckSensor:=FALSE;   step:=step+1;
		END_IF





	11:	IF UnitAConeCrossCount.CV=iAConeCrossCount  THEN
		RowStopperMotorStopDly(In:=FALSE);
		GetDLy(IN:=FALSE);
		step:=step+1;
		ELSIF UnitAConeCrossCount.CV <> iAConeCrossCount  THEN
		tConeChkDly(IN:=TRUE , PT:=t#5s , Q=> , ET=> );

	 (*	IF tConeChkDly.Q THEN bUnitAConeMiss:=TRUE; ELSE bUnitAConeMiss:=FALSE ;  END_IF *)
		END_IF

	12:	IF NOT bAPauseSeq THEN step:=step+1;
		END_IF

	13:	IF bAutoModeOn   THEN
		 UnitAConeCrossCount.RESET:=TRUE;
		step:=step+1;
		END_IF

	14:	UnitAConeCrossCount.RESET:=FALSE; step:=step+1;


	15: 	IF bAutoModeOn AND bIUnitA_RowStopperEnd THEN
		bQAUnitA_RowStopperMotorFwd1:=FALSE;
		tRowStopperRevDly1(IN:=FALSE);
		 step:=step+1;
		ELSIF  bAutoModeOn AND NOT  bIUnitA_RowStopperEnd THEN
		 step:=4;
		END_IF

	16:	step:=step+1;

	17:	tRowStopperRevDly1(IN:=TRUE , PT:=t#1.5s , Q=> , ET=> );
		IF tRowStopperRevDly1.Q THEN step:=step+1; END_IF

	18:	 step:=step+1;


	19:	IF bAutoModeOn   THEN
		bQAUnitA_RowStopperMotorRev1:=TRUE;
		step:=step+1;
		END_IF

	20:	IF bAutoModeOn (*AND bIUnitA_RowStopperMiddle *)  THEN
		tUnitACountDelay1(IN:=FALSE);
		tRowStopperMidDly1(IN:=TRUE , PT:=t#0.2s , Q=> , ET=> );
		IF tRowStopperMidDly1.Q THEN  step:=step+1;
		END_IF
		END_IF


	21:	tUnitACountDelay1(IN:=TRUE , PT:=t#5s , Q=> , ET=> );
		IF tUnitACountDelay1.Q THEN
		step:=step+1;
		END_IF




	22:	IF bAutoModeOn  AND UnitAConeCompChkCount.CV>=iATotalNoOfCones   THEN
		bUnitARowStopperStarted:=FALSE;
		UnitAConeCompChkCount.RESET:=TRUE;
		bStartUnitaCompCount:=FALSE;
		TestTimer(IN:=FALSE);
                  	step:=step+1;
		ELSIF  bAutoModeOn  AND UnitAConeCompChkCount.CV < iATotalNoOfCones  THEN
		TestTimer(IN:=FALSE);
		 ConeInCompleteA:=TRUE;
	(*	ConeInCompletetest:=TRUE; *)
		(*bStartUnitaCompCount:=FALSE;*)
		step:=step+1;

		END_IF


	23:	IF bAutoModeOn AND bIUnitA_RowStopperHome   AND ConeInCompleteA  THEN
		bQAUnitA_RowStopperMotorRev1:=FALSE;
		tRowStopperMidDly1(IN:=FALSE);
		sRetreivalAStatus:= 'IDLE';
		PROCESSCOMPLETE:=TRUE;
		step:=0;
		ELSIF  bAutoModeOn AND bIUnitA_RowStopperHome   AND NOT ConeInCompleteA  THEN
		bQAUnitA_RowStopperMotorRev1:=FALSE;
		tRowStopperMidDly1(IN:=FALSE);
		sRetreivalAStatus:= 'IDLE';

		PROCESSCOMPLETE:=TRUE;
		step:=0;
		END_IF

END_CASE

(***Incomplete Reset**)

IF  bAutoModeOn AND ConeInCompleteA   THEN
TEnableCounter:=TRUE;
ELSE
TEnableCounter:=FALSE;
END_IF



IF  bAutoModeOn AND ConeInCompleteA   AND   UnitAConeCompChkCount.CV >= iATotalNoOfCones THEN
TestTimer(IN:=TRUE , PT:=t#5s , Q=> , ET=> );
CycleComplete:=TRUE;
bStartUnitaCompCount:=FALSE;

END_IF


IF TestTimer.Q THEN
CycleComplete:=FALSE;
UnitAConeCompChkCount.RESET:=TRUE;
bUnitARowStopperStarted:=FALSE;
ConeInCompleteA :=FALSE;
TestTimer(IN:=FALSE);
END_IF
(*

IF  bAutoModeOn AND UnitAConeCompChkCount.CV >= iATotalNoOfCones THEN
TEnableCounter:=FALSE;
tUnitACountDelay1(IN:=FALSE);
ConeInComplete:=FALSE;

END_IF

IF   bAutoModeOn  AND UnitAConeCompChkCount.CV >=iATotalNoOfCones   AND( bUnitARowStopperStarted OR ConeInCompletetest) THEN
CompleteTestbitA:=TRUE;
bStartUnitaCompCount:=FALSE;
UnitAConeCompChkCount.RESET:=TRUE;
ConeInCompletetest:=FALSE;
ELSE
UnitAConeCompChkCount.RESET:=FALSE;
END_IF
*)
UnitAConeCrossCount(
	CU:= bAUnitAConeCrossing_1  (*   R_TRIG_1.Q*) ,
	RESET:= ,
	PV:=12,
	Q=> ,
	CV=> );



UnitAConeCompChkCount(
	CU:=  bAUnitBConeCrossing_1 ,
	RESET:= ,
	PV:=iATotalNoOfCones,
	Q=> ,
	CV=> );
UnitAConeCountHMI:=UnitAConeCompChkCount.CV;
UnitAConeCountHMI_1:=UnitAConeCompChkCount.CV;

(*=======For Retrival A Limit Switch======*)
(*
LimitSwitchBCount(
	CU:=  bAUnitBConeCrossing_1,
	RESET:= ,
	PV:=iATotalNoOfCones,
	Q=> ,
	CV=> );
*)

IF UnitAConeCompChkCount.CV >=  iATotalNoOfCones AND bIUnitA_RowStopperHome  AND NOT bQAUnitA_RowStopperMotorRev1 AND NOT ConeInCompleteA  THEN tConeCrossDly(IN:=TRUE , PT:=t#0.5s , Q=> , ET=> );  END_IF
(*
IF LimitSwitchBCount.CV< iATotalNoOfCones AND bUnitARowStopperStarted THEN  CountAtLimitBNok:=TRUE;ELSE CountAtLimitBNok:=FALSE;  (*CountCheckdly(IN:=TRUE , PT:=t#5s , Q=> , ET=> )*); END_IF*)

IF tConeCrossDly.Q THEN bUnitARowStopperStarted:=FALSE; UnitAConeCompChkCount.RESET:=TRUE; step:=0;  tConeCrossDly(IN:=FALSE); ELSE  UnitAConeCompChkCount.RESET:=FALSE; END_IF

(*
ELSE
UnitAConeCompChkCount.RESET:=FALSE; *)



(*===============Stop Sequence===========*)


IF NOT bIEmergency  OR  bStopHmi  OR bAutoModeOff  OR bIMCStop   THEN bStopRetUnitA:=TRUE; END_IF


IF bStopRetUnitA (*AND NOT  bIUnitA_RowStopperHome *) THEN
ConeInCompleteA:=FALSE;
step:=0;
step2:=0;
step4:=0;
bAUnitAWeighOk:=FALSE;
bQAUnitA_RowStopperMotorFwd1:=FALSE;
bUnitARowStopperStarted:=FALSE;
UnitAConeCrossCount.RESET:=TRUE;
bQAUnitA_RowStopperMotorFwd2:=FALSE;
UnitAConeCompChkCount.RESET:=TRUE;
bQAUnitA_RowStopperMotorRev1:=FALSE;
bRetUnitARst:=TRUE;
bAUnitAConeCrossing_1:=FALSE;
bAUnitBConeCrossing_1:=FALSE;
END_IF

IF bIUnitA_RowStopperHome THEN
bRetUnitARst:=FALSE;
  UnitAConeCompChkCount.RESET:=FALSE;
bStopRetUnitA:=FALSE;
END_IF

(*
(*=============for Pause Operation bypass to Feeding Conveyor==================*)

IF UnitAConeCrossCount.CV >= 1 AND bPauseHmi AND  UnitAConeCrossCount.CV=iAConeCrossCount THEN bPauseExtend:=TRUE; ELSE  bPauseExtend:=FALSE;  END_IF


*)



(*IF NOT CompleteTestbitA THEN  *)
CASE step2 OF

	0:	IF   (bStartUnitaCompCount  (*bUnitARowStopperStarted  *) OR  TEnableCounter  ) THEN
		F_TRIG_3(CLK:=bIUnitBConeCrossing , Q=> );
		IF F_TRIG_3.Q THEN TON_6(IN:= FALSE); step2:=step2+1; END_IF END_IF


	1:	TON_6(IN:= FALSE);
		TON_9(IN:= FALSE);
		step2:=step2+1;


	2:	 bAUnitBConeCrossing_1 :=TRUE;
		 step2:=Step2+1;

	3:	 step2:=step2+1;

	4: 	TON_6(IN:=  TRUE  , PT:=t#100ms,Q=> , ET=> );
		IF TON_6.Q THEN bAUnitBConeCrossing_1:=FALSE;   step2:=step2+1; END_IF


	5:	 step2:=step2+1;

	6:	IF   bIUnitBConeCrossing THEN
		TON_9(IN:=  TRUE  , PT:=t#50ms,Q=> , ET=>);
		IF TON_9.Q THEN TON_6(IN:= FALSE);  step2:=step2+1; END_IF END_IF


	7:	 step2:=step2+1;

	8:	 step2:=step2+1;

	9:	 step2:=step2+1;

	10:	TON_9(IN:= FALSE);
		step2:=0;


END_CASE
(*END_IF *)


CASE step4 OF

	0:	IF bUnitARowStopperStarted THEN
		F_TRIG_5(CLK:=bIUnitAConeCrossing , Q=> );
		IF F_TRIG_5.Q THEN TON_8(IN:= FALSE); step4:=step4+1; END_IF END_IF


	1:	TON_8(IN:= FALSE);
		TON_10(IN:= FALSE);
		step4:=step4+1;


	2:	 bAUnitAConeCrossing_1 :=TRUE;
		 step4:=step4+1;

	3:	 step4:=step4+1;

	4: 	TON_8(IN:=  TRUE  , PT:=t#100ms,Q=> , ET=> );
		IF TON_8.Q THEN  bAUnitAConeCrossing_1:=FALSE;  step4:=step4+1; END_IF


	5:	 step4:=step4+1;

	6:	IF   bIUnitAConeCrossing THEN
		TON_10(IN:=  TRUE  , PT:=t#50ms,Q=> , ET=>);
		IF TON_10.Q THEN TON_8(IN:= FALSE);  step4:=step4+1; END_IF END_IF


	7:	 step4:=step4+1;;

	8:	 step4:=step4+1;

	9:	 step4:=step4+1;

	10:	TON_8(IN:= FALSE);
		step4:=0;


END_CASE


IF bRetUnitAStart THEN step4:=0; step2:=0 ; END_IF
END_PROGRAM

(* POU FunctionBlocks/SenSelect, ST *)
FUNCTION_BLOCK SenSelect
VAR_INPUT


	bVarIn1: BOOL;
	bVarIn2: BOOL;
	bVarIn3: BOOL;
	bVarIn4: BOOL;
END_VAR
VAR_OUTPUT


	ByteResult: USINT;
END_VAR
VAR

END_VAR
ByteResult.0:=bVarIn1;
ByteResult.1:=bVarIn2;
ByteResult.2:=bVarIn3;
ByteResult.3:=bVarIn4;

ByteResult;
END_FUNCTION_BLOCK

(* POU AutoMode/UnitB_RowStopper, ST *)
PROGRAM UnitB_RowStopper
VAR
	step: INT;
	bAUnitAWeighOk: BOOL;
	CTU_1: CTU;
	CTU_1Enable: BOOL;
	R_TRIG_1: R_TRIG;
	R_TRIG_2: F_TRIG;
	bQAUnitA_RowStopperMotorFwd1: BOOL;
	bQAUnitA_RowStopperMotorFwd2: BOOL;
	tRowStopperRevDly1: TON;
	bQAUnitA_RowStopperMotorRev1: BOOL;
	CTU_2: CTU;
	UnitBConeCount: CTU;
	CTU_1EnableUnitB: BOOL;
	temp1: BOOL;
	bStopRetUnitB: BOOL;
	bRetUnitBRst: BOOL;
	RowStopperMotorStopDly: TON;
	F_TRIG_3: F_TRIG;
	UnitBCompleteCheckCount:CTU;
	UnitBOverTemp: BOOL;
	bStartTemp1: BOOL;
	R_TRIG_5: R_TRIG;
	test: BOOL;
	bStopTemp2: BOOL;
	CTU_2CV: INT;
	CTU_test: CTU;
	R_TRIG_test: R_TRIG;
	InterLockStep: INT;

	CTU_2Enable: BOOL;
	timer1: TON;
	UnitBCompleteCheckCountCV: INT;
	Ctu_2_Rst: BOOL;
	F_TRIG_1: F_TRIG;
	bRestBit: BOOL;
	bResetBit: BOOL;
	R_TRIG_6: R_TRIG;
	timer2: TON;
	UnitBConeCrossCount: CTU;
	bQAUnitB_RowStopperMotorFwd1: BOOL;
	sRetreivalBStatus: STRING;
	GetDLy: TON;
	bCheckSensor: BOOL;
	iAConeCrossCount: INT;
	bQAUnitB_RowStopperMotorRev1: BOOL;
	iSensorOnVal: USINT;
	SenSelect_2: SenSelect;
	tConeChkDly: TON;
	bConeMiss: BOOL;
	tConeCrossDly: TON;
	UnitBConeCompChkCount: CTU;
	iAConeCrossPVal: INT;
	TON_6: TON;
	step2: INT;
	bAUnitBConeCrossing_1: BOOL;
	bAUnitBConeCrossedOff: BOOL;
	R_TRIG_3: R_TRIG;
	TON_8: TON;
	R_TRIG_11: R_TRIG;

	F_TRIG_4: F_TRIG;
	tRowStopperMidDly2: TON;
	tUnitBCountDelay1: TON;

	TEnableCounterB: BOOL;
	CompleteTestbitB: BOOL;
	bCounterDisableUnitB: BOOL;
	TestTimer: TON;
	bStartUnitBCompCount: BOOL;
	step3: INT;
	F_TRIG_5: F_TRIG;
	TON_9: TON;
	TON_10: TON;
	TON_11: TON;
	TON_12: TON;
	bAUnitBConeCrossedTemp: BOOL;
END_VAR
(*=============CHecking the No of sensors sensed on conveyor ==================*)

IF bCheckSensor THEN
SenSelect_2(
		bVarIn1:=bIUnitBConeDetection1 ,
		bVarIn2:= bIUnitBConeDetection2,
		bVarIn3:= bIUnitBConeDetection3,
		bVarIn4:= bIUnitBConeDetection4,
		ByteResult=>iSensorOnVal );


END_IF

IF iSensorOnVal=15 THEN iAConeCrossCount:=4;
		ELSIF  iSensorOnVal=14 THEN iAConeCrossCount:=3;
		ELSIF  iSensorOnVal=13 THEN iAConeCrossCount:=3;
		ELSIF  iSensorOnVal=12 THEN iAConeCrossCount:=2;
		ELSIF  iSensorOnVal=11 THEN iAConeCrossCount:=3;
		ELSIF  iSensorOnVal=10 THEN iAConeCrossCount:=2;
		ELSIF  iSensorOnVal=9 THEN iAConeCrossCount:=2;
		ELSIF  iSensorOnVal=8 THEN iAConeCrossCount:=1;
		ELSIF  iSensorOnVal=7 THEN iAConeCrossCount:=3;
		ELSIF  iSensorOnVal=6 THEN iAConeCrossCount:=2;
		ELSIF  iSensorOnVal=5 THEN iAConeCrossCount:=2;
		ELSIF  iSensorOnVal=4 THEN iAConeCrossCount:=1;
		ELSIF  iSensorOnVal=3 THEN iAConeCrossCount:=2;
		ELSIF  iSensorOnVal=2 THEN iAConeCrossCount:=1;
		ELSIF  iSensorOnVal=1 THEN iAConeCrossCount:=1;
		END_IF





bQAUnitBRowStopperMotorFwd:=( bQAUnitB_RowStopperMotorFwd1  );

bQAUnitBRowStopperMotorRev:= ( bQAUnitB_RowStopperMotorRev1 OR bRetUnitBRst  );

CASE step OF

	0:	CycleComplete1:=FALSE;
		IF bAutoModeOn  AND bAUnitBWeighOk  AND bRetUnitBStart  AND NOT bAInializeStarted AND NOT bIntialAckBit AND bInterlockInitial_2  THEN
		UnitBConeCrossCount.RESET:=TRUE;

		CTU_2.RESET:=TRUE;
		step:=step+1;
		END_IF

	1:
		PROCESSCOMPLETE:=FALSE;step:=step+1;

	2:	IF bAutoModeOn(* AND bIUnitB_LiftPistonHome *)THEN
		CTU_2.RESET:=FALSE;
		UnitBConeCrossCount.RESET:=FALSE;
		UnitBCompleteCheckCount.RESET:=FALSE;
		step:=step+1;
		END_IF


	3:	UnitBConeCompChkCount.RESET:=FALSE;
		TestTimer(IN:=FALSE);
		step:=step+1;


	4:	IF bAutoModeOn   AND NOT  bUnitARowStopperStarted  AND NOT ConeInCompleteA AND NOT  ConeInCompleteB  AND NOT bAPauseSeq
		(*AND NOT bIUnitBConedetection1 AND NOT bIUnitBConedetection2 AND NOT bIUnitBConedetection3 *) AND bInterlockInitial_2 THEN
		timer1(IN:=FALSE);
		timer2(IN:=FALSE);
		bQAUnitB_RowStopperMotorFwd1:=TRUE;
		bAUnitBWeighOk:=FALSE;
		sRetreivalBStatus:= 'Running';
		bUnitBRowStopperStarted:=TRUE;
	(*	UnitBConeCrossCount.RESET:=TRUE; *)

		step:=step+1;
		END_IF

	5:	RowStopperMotorStopDly(In:=FALSE); step:=step+1;


	6:	IF bIUnitBConedetection1 OR  bIUnitBConedetection2  OR  bIUnitBConedetection3  OR bIUnitBConedetection4  AND NOT bAPauseSeq THEN

		step:=step+1;
		ELSIF NOT bIUnitBConedetection1 AND NOT  bIUnitBConedetection2 AND NOT  bIUnitBConedetection3 AND NOT bIUnitBConedetection4  AND bIUnitB_RowStopperEnd THEN

		step:=15;

		END_IF

	7:	CompleteTestbitB:=FALSE;
		UnitBConeCompChkCount.RESET:=TRUE;
		RowStopperMotorStopDly( IN:=TRUE , PT:=T#0.4S , Q=> , ET=> );
		IF RowStopperMotorStopDly.Q   THEN UnitBConeCrossCount.RESET:=FALSE;  UnitBConeCompChkCount.RESET:=FALSE ; step:=step+1; END_IF


	8:	bStartUnitBCompCount:=TRUE;
		bQAUnitB_RowStopperMotorFwd1:=FALSE;
		tRowStopperRevDly1(IN:=FALSE);
		GetDLy(IN:=FALSE);
		step:=step+1;

	9:	IF NOT   bAPauseSeq THEN bCheckSensor:=TRUE; step:=step+1;END_IF

	10:	GetDLy(IN:=TRUE , PT:=t#0.4s , Q=> , ET=> );
		 IF GetDLy.Q THEN bCheckSensor:=FALSE;  tConeChkDly(IN:=FALSE);  step:=step+1;
		END_IF



	11:	IF UnitBConeCrossCount.CV>=iAConeCrossCount  THEN
		RowStopperMotorStopDly(In:=FALSE);
		 tConeChkDly(IN:=FALSE);
		GetDLy(IN:=FALSE);
		step:=step+1;
		ELSIF UnitBConeCrossCount.CV <> iAConeCrossCount  THEN
		tConeChkDly(IN:=TRUE , PT:=t#5s , Q=> , ET=> );
	(*	IF tConeChkDly.Q THEN bConeMiss:=TRUE; ELSE bConeMiss:=FALSE ;  END_IF *)
		END_IF


	12:	IF NOT bAPauseSeq THEN tRowStopperRevDly1(IN:=FALSE); step:=step+1; END_IF

	13:	IF bAutoModeOn   THEN
		UnitBConeCrossCount.RESET:=TRUE;
		step:=step+1;
		END_IF


	14:	 UnitBConeCrossCount.RESET:=FALSE; step:=step+1;

	15:	IF bAutoModeOn AND bIUnitB_RowStopperEnd THEN
		bQAUnitB_RowStopperMotorFwd1:=FALSE;
		 step:=step+1;
		ELSIF  bAutoModeOn AND NOT  bIUnitB_RowStopperEnd  THEN
		 step:=4;
		END_IF

	16:	tRowStopperRevDly1(IN:=TRUE , PT:=t#1.5s , Q=> , ET=> );
		IF tRowStopperRevDly1.Q THEN step:=step+1; END_IF

	17:	step:=step+1;

	18:	IF bAutoModeOn THEN
		tRowStopperMidDly2(IN:=FALSE);
		UnitBConeCount.RESET:=FALSE;
		bQAUnitB_RowStopperMotorRev1:=TRUE;
		step:=step+1;
		END_IF

	19:	IF bAutoModeOn (*AND bIUnitB_RowStopperMiddle*)   THEN
		  tUnitBCountDelay1(IN:=FALSE);
		tRowStopperMidDly2(IN:=TRUE , PT:=t#0.2s , Q=> , ET=> );
		IF tRowStopperMidDly2.Q THEN   bCounterDisableUnitB:=TRUE;  step:=step+1;
		END_IF
		END_IF

	20:    tUnitBCountDelay1(IN:=TRUE , PT:=t#5s , Q=> , ET=> );
		IF tUnitBCountDelay1.Q THEN CycleComplete1:=TRUE; step:=step+1; END_IF

	21:	IF bAutoModeOn  AND UnitBCompleteCheckCount.CV >=iATotalNoOfCones THEN
		bUnitBRowStopperStarted:=FALSE;
		(*UnitBCompleteCheckCount.RESET:=TRUE;*)
	(*	bUnitACounterDIsable:=TRUE; *)
		bStartUnitBCompCount:=FALSE;
		step:=step+1;
		ELSIF  bAutoModeOn  AND UnitBCompleteCheckCount.CV < iATotalNoOfCones  THEN
		ConeInCompleteB:=TRUE;
		(*bStartUnitBCompCount:=FALSE;*)
		step:=step+1;
		END_IF

	22:	IF bAutoModeOn AND bIUnitB_RowStopperHome  AND ConeInCompleteB THEN
		bQAUnitB_RowStopperMotorRev1:=FALSE;
		tRowStopperMidDly2(IN:=FALSE);
		sRetreivalBStatus:= 'IDLE';
		step:=step+1;
		ELSIF bAutoModeOn AND bIUnitB_RowStopperHome  AND NOT ConeInCompleteB THEN
		bQAUnitB_RowStopperMotorRev1:=FALSE;
		tRowStopperMidDly2(IN:=FALSE);
		sRetreivalBStatus:= 'IDLE';
		PROCESSCOMPLETE:=TRUE;
		step:=step+1 (*step+1*);
		END_IF

	23:	IF bAutoModeOn  AND UnitBCompleteCheckCount.CV >=iATotalNoOfCones THEN
		bUnitBRowStopperStarted:=FALSE;
		UnitBCompleteCheckCount.RESET:=TRUE;
		step:=step+1;
		END_IF

	24:	ConeInCompleteB :=FALSE;step:=0;


END_CASE
(***Incomplete Reset**)

IF  bAutoModeOn AND ConeInCompleteB   THEN
TEnableCounterB:=TRUE;
ELSE
TEnableCounterB:=FALSE;
(*bUnitBRowStopperStasrted:=FALSE; *)
END_IF

IF  bAutoModeOn AND ConeInCompleteB   AND   UnitBCompleteCheckCount.CV >=iATotalNoOfCones   THEN
TestTimer(IN:=TRUE , PT:=t#5s , Q=> , ET=> );

END_IF

IF TestTimer.Q THEN
CycleComplete1:=FALSE;
(*UnitBCompleteCheckCount.RESET:=TRUE;*)
bUnitBRowStopperStarted:=FALSE;
ConeInCompleteB :=FALSE;
TestTimer(IN:=FALSE);
bStartUnitBCompCount:=FALSE;
END_IF

(*
IF bAutoModeOn  AND    bCounterDisableUnitB  AND   UnitBCompleteCheckCount.CV >=iATotalNoOfCones AND( bUnitBRowStopperStarted OR ConeInCompleteTestbitB) THEN
CompleteTestbitB:=TRUE;
bStartUnitBCompCount:=FALSE;
UnitBCompleteCheckCount.RESET:=TRUE;
ConeInCompleteTestbitB:=FALSE;
bCounterDisableUnitB:=FALSE;
ELSE
UnitBCompleteCheckCount.RESET:=FALSE;
END_IF
*)





(*F_TRIG_11(CLK:=bIUnitBConeCrossing , Q=> ); *)
UnitBConeCrossCount(
	CU:=  bAUnitBConeCrossedTemp ,
	RESET:= ,
	PV:=3 ,
	Q=> ,
	CV=> );
(*
UnitBConeCompChkCount(
	CU:= bIUnitBConeCrossing  (*   R_TRIG_1.Q*) ,
	RESET:= ,
	PV:=50,
	Q=> ,
	CV=> );
*)


(*=Total Cone crossing the Unit B Limit Switch==========*)

UnitBCompleteCheckCount(
	CU:=   bAUnitBConeCrossed  ,
	RESET:= ,
	PV:=iATotalNoOfCones ,
	Q=> ,
	CV=>UnitBCompleteCheckCountCV );

UnitBConeCountHMI:=UnitBCompleteCheckCount.CV;

IF UnitBCompleteCheckCount.CV >=  iATotalNoOfCones  AND bIUnitB_RowStopperHome  AND NOT bQAUnitB_RowStopperMotorRev1 AND NOT ConeInCompleteB THEN
 tConeCrossDly(IN:=TRUE , PT:=t#0.5s , Q=> , ET=> );
END_IF

IF tConeCrossDly.Q THEN
 bUnitBRowStopperStarted:=FALSE;
UnitBCompleteCheckCount.RESET:=TRUE;
step:=0;
  tConeCrossDly(IN:=FALSE);
ELSE
UnitBCompleteCheckCount.RESET:=FALSE;

END_IF






(*===============Stop Sequence===========*)


IF NOT  bIEmergency OR   bStopHmi OR bAutoModeOff  OR bIMCStop  THEN bStopRetUnitB:=TRUE;
(*
b12ConeModelSelected:=FALSE;
b18ConeModelSelected:=FALSE;
b24ConeModelSelected:=FALSE;
b32ConeModelSelected:=FALSE;

iNetWtHmi:=0;
iNetTolHmi:=0;
rSealCompDlyHmi:=0;
*)
NegToleranceEnabled:=TRUE; UnitBCompleteCheckCount.RESET:=TRUE;
END_IF


IF bStopRetUnitB  (*AND NOT bIUnitB_RowStopperHome *) THEN
ConeInCompleteB:=FALSE;
step:=0;
step2:=0;
bAUnitBWeighOk:=FALSE;
bAUnitBConeCrossed:=FALSE;
bQAUnitB_RowStopperMotorFwd1:=FALSE;
UnitBConeCount.RESET:=TRUE;
UnitBCompleteCheckCount.RESET:=TRUE;
bQAUnitB_RowStopperMotorRev1:=FALSE;
bRetUnitBRst:=TRUE;
bUnitBRowStopperStarted:=FALSE;
UnitBCompleteCheckCount.RESET:=TRUE;
TON_6(IN:= FALSE);
TON_8(IN:= FALSE);
TON_9(IN:= FALSE);
TON_10(IN:= FALSE);
END_IF

IF bIUnitB_RowStopperHome THEN
bStopRetUnitB:=FALSE;
bRetUnitBRst:=FALSE;

END_IF

(*IF NOT CompleteTestbitB THEN  *)
CASE step2 OF

	0:	IF bStartUnitBCompCount (* bUnitBRowStopperStarted *)OR TEnableCounterB THEN
		F_TRIG_4(CLK:=bIUnitBConeCrossing , Q=> );
		IF F_TRIG_4.Q THEN TON_6(IN:= FALSE); step2:=step2+1; END_IF END_IF


	1:	TON_6(IN:= FALSE);
		TON_8(IN:= FALSE);
		step2:=step2+1;


	2:	 bAUnitBConeCrossed:=TRUE;
		 step2:=Step2+1;

	3:	 step2:=step2+1;

	4: 	TON_6(IN:=  TRUE  , PT:=t#50ms,Q=> , ET=> );
		IF TON_6.Q THEN  bAUnitBConeCrossed:=FALSE;  step2:=step2+1; END_IF


	5:	 step2:=step2+1;

	6:	IF  bIUnitBConeCrossing THEN
		TON_6(IN:= FALSE);
		step2:=step2+1; END_IF

	7:	TON_8(IN:=  TRUE  , PT:=t#10ms,Q=> , ET=> );
		IF TON_8.Q THEN  step2:=step2+1; END_IF

	8:	 step2:=step2+1;

	9:	 step2:=step2+1;

	10:	TON_8(IN:= FALSE);
		step2:=0;


END_CASE
(*END_IF  *)






IF bAutoModeOn  AND  bResetBit AND bIUnitBConedetection1 AND bIUnitBConedetection3 AND bIUnitBConedetection3    AND NOT  bIUnitB_RowStopperHome THEN Ctu_2_Rst:=TRUE;  ELSE Ctu_2_Rst:= FALSE; END_IF

R_TRIG_6(CLK:=Ctu_2_Rst , Q=> );

CTU_2.RESET:= R_TRIG_6.Q;

CASE step3 OF

	0:	IF bStartUnitBCompCount THEN
		F_TRIG_5(CLK:=bIUnitBConeCrossing , Q=> );
		IF F_TRIG_5.Q THEN TON_9(IN:= FALSE); step3:=step3+1; END_IF END_IF


	1:	TON_9(IN:= FALSE);
		TON_10(IN:= FALSE);
		step3:=step3+1;


	2:	 bAUnitBConeCrossedTemp:=TRUE;
		 step3:=Step3+1;

	3:	 step3:=step3+1;

	4: 	TON_11(IN:=  TRUE  , PT:=t#50ms,Q=> , ET=> );
		IF TON_11.Q THEN  bAUnitBConeCrossedTemp:=FALSE;  step3:=step3+1; END_IF


	5:	 step3:=step3+1;

	6:	IF  bIUnitBConeCrossing THEN
		TON_11(IN:= FALSE);
		step3:=step3+1; END_IF

	7:	TON_12(IN:=  TRUE  , PT:=t#10ms,Q=> , ET=> );
		IF TON_12.Q THEN  step3:=step3+1; END_IF

	8:	 step3:=step3+1;

	9:	 step3:=step3+1;

	10:	TON_12(IN:= FALSE);
		step3:=0;


END_CASE
END_PROGRAM

(* POU Manual/Manual, ST *)
PROGRAM Manual
VAR
	b_SHPistonValveREVOffHmi: BOOL;
	Timer1: TON;
	step: INT;
	bIManualSealingTemp: BOOL;
	bEnableManSeal1: BOOL;
	bEnableManSeal2: BOOL;
	bEnableManSeal: BOOL;
END_VAR
(*=============MANUAL OPERATION============*)



(*=============UNIT-A ROW STOPPER MOTOR FWD & REV==========*)


	IF  bManualModeOn AND  bUA_RowStopperMotorFwdOnHmi  AND NOT bIUnitA_RowStopperEnd    THEN	bQMUnitA_RowStopperMotorForward:=TRUE; ELSE   bQMUnitA_RowStopperMotorForward:=FALSE; END_IF
	IF  bManualModeOn AND   bIUnitA_RowStopperEnd THEN bQMUnitA_RowStopperMotorForward:=FALSE; END_IF




	IF bManualModeOn AND bUA_RowStopperMotorRevOnHmi AND NOT bIUnitA_RowStopperHome THEN	bQMUnitA_RowStopperMotorReverse:=TRUE; ELSE  bQMUnitA_RowStopperMotorReverse:=FALSE;  END_IF
	IF  bManualModeOn AND   bIUnitA_RowStopperHome THEN  bQMUnitA_RowStopperMotorReverse:=FALSE;  END_IF



(*=============UNIT-B ROW STOPPER MOTOR FWD & REV==========*)


	IF  bManualModeOn AND  bUB_RowStopperMotorFwdOnHmi AND NOT  bIUnitB_RowStopperEnd   THEN	bQMUnitB_RowStopperMotorForward:=TRUE; ELSE  	bQMUnitB_RowStopperMotorForward:=FALSE;   END_IF
	IF  bManualModeOn AND   bIUnitB_RowStopperEnd THEN bQMUnitB_RowStopperMotorForward:=FALSE; END_IF




	IF bManualModeOn AND bUB_RowStopperMotorRevOnHmi  AND NOT   bIUnitB_RowStopperHome   THEN 	bQMUnitB_RowStopperMotorReverse:=TRUE; ELSE  bQMUnitB_RowStopperMotorReverse:=FALSE;    END_IF
	IF  bManualModeOn AND   bIUnitB_RowStopperHome THEN  bQMUnitB_RowStopperMotorReverse:=FALSE;  END_IF




(**************************CONE FEEDING OPERATION***************************)

	IF bManualModeOn AND bCFPistonOnHmi THEN bQMConeFeedingPistonValve:=TRUE; END_IF
	IF bManualModeOn AND bCFPistonOffHmi THEN bQMConeFeedingPistonValve:=FALSE;END_IF

(*=============FORWARD PISTON VALVE=================*)

	IF bManualModeOn AND bFPValveOnHmi  THEN bQMForwardPistonValve:=TRUE;END_IF
	IF bManualModeOn AND bFPValveOffHmi THEN bQMForwardPistonValve:=FALSE;END_IF


(*=================WRAPPING CHANNEL1=================*)

	IF bManualModeOn AND bWrappingCPV1OnHmi THEN bQMWrappingChannelPistonValve1:=TRUE;END_IF
	IF bManualModeOn AND bWrappingCPV1OffHmi THEN bQMWrappingChannelPistonValve1:=FALSE;END_IF


(*=================WRAPPING CHANNEL2=================*)

	IF bManualModeOn AND bWrappingCPV2OnHmi THEN bQMWrappingChannelPistonValve2:=TRUE;END_IF
	IF bManualModeOn AND bWrappingCPV2OffHmi THEN bQMWrappingChannelPistonValve2:=FALSE;END_IF

(*=================WRAPPING CHANNEL3=================*)

	IF bManualModeOn AND bWrappingCPV3OnHmi THEN bQMWrappingChannelPistonValve3:=TRUE;END_IF
	IF bManualModeOn AND bWrappingCPV3OffHmi THEN bQMWrappingChannelPistonValve3:=FALSE;END_IF

(*=================SEALING TOP PISTON=================*)

	IF bManualModeOn AND bSealingTopPVOnHmi THEN bQMSealingTopPistonValve:=TRUE;END_IF
	IF bManualModeOn AND bSealingTopPVOffHmi THEN bQMSealingTopPistonValve:=FALSE;END_IF

(*=================SEALING BOTTOM PISTON=================*)

	IF bManualModeOn AND bSealingBottomPVOnHmi	 THEN bQMSealingBottomPistonValve:=TRUE;END_IF
	IF bManualModeOn AND bSealingBottomPVOffHmi THEN bQMSealingBottomPistonValve:=FALSE;END_IF

(*=================FEEDING CONVEYOR MOTOR=================*)

	IF  bManualModeOn AND       bFCMotorOnHmi THEN bQMFeedingConveyorMotor:=TRUE;END_IF
	IF   bManualModeOn AND      bFCMotorOffHmi THEN bQMFeedingConveyorMotor:=FALSE;END_IF

(*=================WRAPPING CONVEYOR MOTOR=================*)

	IF bManualModeOn AND bWCMotorOnHmi THEN bQMWrappingConveyorMotor:=TRUE;END_IF
	IF bManualModeOn AND bWCMotorOffHmi THEN bQMWrappingConveyorMotor:=FALSE;END_IF

(*=================SEALING CONVEYOR MOTOR=================*)

	IF bManualModeOn AND bSCMotorOnHmi THEN bQMSealingConveyorMotor:=TRUE;END_IF
	IF bManualModeOn AND bSCMotorOffHmi THEN bQMSealingConveyorMotor:=FALSE;END_IF

(*=================FLIM ROLLER MOTOR1=================*)

	IF bManualModeOn AND bFRMotor1OnHmi THEN bQMFilmRollerMotor1:=TRUE;END_IF
	IF bManualModeOn AND bFRMotor1OffHmi THEN bQMFilmRollerMotor1:=FALSE;END_IF

(*=================FLIM ROLLER MOTOR2=================*)

	IF bManualModeOn AND bFRMotor2OnHmi THEN bQMFilmRollerMotor2:=TRUE;END_IF
	IF bManualModeOn AND bFRMotor2OffHmi THEN bQMFilmRollerMotor2:=FALSE;END_IF

(*=================FLIM ROLLER MOTOR3=================*)

	IF bManualModeOn AND bFRMotor3OnHmi THEN bQMFilmRollerMotor3:=TRUE;END_IF
	IF bManualModeOn AND bFRMotor3OffHmi THEN bQMFilmRollerMotor3:=FALSE;END_IF

(*==============SEALING SEPARATOR Y PISTON VALVE===================*)

	IF bManualModeOn AND bSSYAxisPistonValveOnHmi THEN  bQMSealingSeparatorYAxisPistonValve:=TRUE;END_IF
	IF bManualModeOn AND bSSYAxisPistonValveOffHmi THEN  bQMSealingSeparatorYAxisPistonValve:=FALSE;END_IF


(*================SEALING SEPARATOR X PISTON VALVE=================*)

	IF bManualModeOn AND bSSXAxisPistonValveOnHmi THEN  bQMSealingSeparatorXAxisPistonValve:=TRUE;END_IF
	IF bManualModeOn AND bSSXAxisPistonValveOffHmi THEN  bQMSealingSeparatorXAxisPistonValve:=FALSE;END_IF







(*======================manual Sealing Logic==========================*)

IF NOT bAutoModeOn AND bIManualSealing THEN bEnableManSeal1:=TRUE; ELSE  bEnableManSeal1:=FALSE; END_IF

 IF bAutoModeOn AND bIManualSealing AND bAPauseSeq  THEN bEnableManSeal2:=TRUE; ELSE  bEnableManSeal2:=FALSE; END_IF

IF bEnableManSeal1 OR bEnableManSeal2 THEN bEnableManSeal:=TRUE; ELSE  bEnableManSeal:=FALSE; END_IF

CASE step OF

	0:	IF bEnableManSeal  THEN bMManualSealOn:=TRUE; step:=step+1;  END_IF

	1:	Timer1(IN:= FALSE);
		bQMSealingTopPistonValve:=TRUE;
		step:=step+1;

	2:	 IF bISealingBottomPistonEnd AND bISealingTopPistonEnd THEN
		 step:=step+1;
		END_IF

	3:	Timer1(IN:=TRUE , PT:=SealComDlyTemp , Q=> , ET=> );
		IF Timer1.Q THEN step:=step+1; END_IF


	4:	bMManualSealOn:=FALSE;
		bQMSealingTopPistonValve:=FALSE;
		Timer1(IN:= FALSE);
		 step:=step+1;

	5:	step:=0;

END_CASE
END_PROGRAM

(* POU Outputs, ST *)
PROGRAM Outputs
VAR
	bQABuzzertemp: BOOL;
END_VAR
		bQConeFeedingPistonValve   :=   (bQMConeFeedingPistonValve OR bQAConeFeedingPistonValve) ;
		bQForwardPistonValve  :=   (bQMForwardPistonValve OR bQAForwardPistonValve OR bQRForwardPistonValve ) ;
		bQWrappingChannelPistonValve1  :=  bQMWrappingChannelPistonValve1 OR  bQAWrappingChannelPistonValve1 OR bQRWrappingChannelPistonValve1;
		bQWrappingChannelPistonValve2  :=  bQMWrappingChannelPistonValve2 OR bQAWrappingChannelPistonValve2 OR bQRWrappingChannelPistonValve2;
		bQWrappingChannelPistonValve3  :=  bQMWrappingChannelPistonValve3 OR bQAWrappingChannelPistonValve3 OR bQRWrappingChannelPistonValve3;
		bQSealingTopPistonValve  :=  bQMSealingTopPistonValve OR bQASealingTopPistonValve OR bQRSealingTopPistonValve ;
		bQSealingBottomPistonValve  :=  bQMSealingBottomPistonValve OR bQASealingBottomPistonValve  ;
		bQSealingSeparatorYAxisPistonValve:=  (bQMSealingSeparatorYAxisPistonValve OR bQASealingSeparatorYAxisPistonValve OR bQRSealingSeparatorYAxisPistonValve );

		bQSealingSeparatorXAxisPistonValve:=  ( bQMSealingSeparatorXAxisPistonValve OR bQASealingSeparatorXAxisPistonValve OR bQRSealingSeparatorXAxisPistonValve );
		bQFeedingConveyorMotor:=bQMFeedingConveyorMotor OR bQAFeedingConveyorMotor  ;
		bQWrappingConveyorMotor:=bQMWrappingConveyorMotor OR bQAWrappingConveyorMotor OR bQRWrappingConveyorMotor;
		bQFilmRollerMotor1:=bQMFilmRollerMotor1 OR bQAFilmRollerMotor1;
		bQFilmRollerMotor2 :=bQMFilmRollerMotor2 OR bQAFilmRollerMotor2;
		bQFilmRollerMotor3 :=bQMFilmRollerMotor3 OR bQAFilmRollerMotor3;
		bQSealingConveyorMotorFWD :=bQMSealingConveyorMotor OR bQASealingConveyorMotor OR bQRSealingConveyorMotor;

		bQUnitARowStopperMotorFwd:=  (bQAUnitARowStopperMotorFwd   OR bQMUnitA_RowStopperMotorForward);
		bQUnitARowStopperMotorRev:= (bQAUnitARowStopperMotorRev OR bQMUnitA_RowStopperMotorReverse  );
		bQUnitBRowStopperMotorFwd:=bQAUnitBRowStopperMotorFwd OR bQMUnitB_RowStopperMotorForward ;
		bQUnitBRowStopperMotorRev :=bQAUnitBRowStopperMotorRev OR bQMUnitB_RowStopperMotorReverse ;
		bQUnitAWeightokLamp:= bQAUnitAWeightokLamp;
		bQUnitAWeightNokLamp:= bQAUnitAWeightNokLamp;
		bQUnitBWeightOkLamp:= bQAUnitBWeightOkLamp;
		bQUnitBWeightNokLamp:= bQAUnitBWeightNokLamp;
		bQTLGreen:=bQAGreen;
		bQTLAmber:=bQAAmber;
		bQTLRed:=bQARed;
		 bQBuzzer:= bQABuzzer;





bQAUnitARowStopperMotorFwd:= bQAUnitA_RowStopperMotorForward1;

bQAUnitARowStopperMotorRev:=bQAUnitA_RowStopperMotorReverse1;
END_PROGRAM

(* POU AutoMode/ConeFeedPiston, ST *)
PROGRAM ConeFeedPiston
VAR

	R_TRIG_1: R_TRIG;
	CounterTiltRst: BOOL;
	step: INT;

	ConeFeedConvFwdDly1: TON;
	CounterTilt23Rst: BOOL;
	CounterTilt23Rst_R_TRIG: R_TRIG;

	bAConeFeedFwdStart23: BOOL;
	CTU_1: CTU;
	test: BOOL;
	CounterTilt23Enable: BOOL;

	CounterTilt23Rst_TRIG: R_TRIG;
	bQAConeFeedingPistonOnAuto1: BOOL;
	bIForwardPistonHometemp: BOOL;
	bIReversePistonHometemp: BOOL;
	bITiltingEndtemp: BOOL;
	bITiltingHometemp: BOOL;


	bErrorCheckBit1: BOOL;

	tFwdRSErrCheckDly: TON;

	FwdRevCylHomeSenOk: BOOL;
	FwdRevCylHomeSenErr: BOOL;
	testtemp: BOOL;
	Timer1: TON;
	bAConeFeedCylReady: BOOL;
	bAConeFeedCylReady1: BOOL;
	bAConeFeedCylReady2: BOOL;
	bAConeFeedCylReady3: BOOL;
	bAConeFeedCylReady4: BOOL;
END_VAR
(*==================== Cone Feeding Piston Logic For 2*3 Model==================*)




		IF   bAutoModeOn AND ConeFeedConvFwdDly1.Q  AND bIConeFeedingPistonHome   AND bIForwardPistonHome   AND  NOT bAPauseSeq AND bAConeFeedCylReady       THEN
		bQAConeFeedingPistonOnAuto1:=TRUE;
		END_IF

		IF    bQAConeFeedingPistonValve AND bAutoModeOn AND  bIConeFeedingPistonEnd AND  NOT bAPauseSeq  AND NOT bAConeFeedCylRsError THEN
		bQAConeFeedingPistonOnAuto1:=FALSE;
		bAConeFeedOver:=TRUE;
		bAConeFeedCylReady1:=FALSE;
		bAConeFeedCylReady2:=FALSE;
		bAConeFeedCylReady3:=FALSE;
		bAConeFeedCylReady4:=FALSE;

		END_IF


(*R_TRIG_1(CLK:= bIConeOrientationTop , Q=> ); *)

ConeFeedConvFwdDly1(IN:=bIConeOrientationTop , PT:=t#0.1s , Q=> , ET=> );  (* ===old Value  PT:=t#1s *)

(*=============Output============*)

bQAConeFeedingPistonValve:=bQAConeFeedingPistonOnAuto1;

bAConeFeedCylReady:= (bAConeFeedCylReady1 OR bAConeFeedCylReady2 OR bAConeFeedCylReady3 OR bAConeFeedCylReady4 );

CASE step OF

	0:	 IF bWrpConvIntOver AND bSealConvIntOver THEN bAConeFeedCylReady1:=TRUE; step:=step+1;  END_IF

	1:	IF bAFwdPistonComp1 THEN bAConeFeedCylReady2:=TRUE; bAFwdPistonComp1:=FALSE;  step:=step+1;  END_IF

	2:	IF bAFwdPistonComp2 THEN bAConeFeedCylReady3:=TRUE;  bAFwdPistonComp2:=FALSE;	 step:=step+1;  END_IF

	3:	IF bAFwdPistonComp3 THEN bAConeFeedCylReady4:=TRUE; bAFwdPistonComp3:=FALSE;	 step:=1;  END_IF





END_CASE

	IF  NOT  bIEmergency   OR bAutoModeOff  OR  bStopHmi OR bIMCStop THEN
	bQAConeFeedingPistonOnAuto1:=FALSE;
	bAFwdPistonComp1:=FALSE;
	bAFwdPistonComp2:=FALSE;
	bAFwdPistonComp3:=FALSE;
	 bAConeFeedOver:=FALSE;
	bWrpConvIntOver:=FALSE;
	bAConeFeedCylReady1:=FALSE;
	bAConeFeedCylReady2:=FALSE;
	bAConeFeedCylReady3:=FALSE;
	bAConeFeedCylReady4:=FALSE;
	ConeFeedConvFwdDly1(IN:=FALSE);

	step:=0;
 END_IF
END_PROGRAM

(* POU AutoMode/ConeFeedConv, ST *)
PROGRAM ConeFeedConv
VAR
	bARetUnitRunning: BOOL;
	bConePresentInConv: BOOL;
	tConeFeedConvStopDly: TON;
	step: INT;
	TON_1: TON;
	TON_2: TON;
	TON_3: TON;
	CTU_2: CTU;
	R_TRIG_2: R_TRIG;
	CTU_2Enable: BOOL;
	TON_4: TON;


	R_TRIG_1: R_TRIG;
	TON_5: TON;
	AllOutputsOn: BOOL;
	bAConveStartsAuto: BOOL;
	R_TRIG_3: R_TRIG;
	TON_6: TON;
	bAUnitBConeCrossingOff: BOOL;
	step2: INT;
	testCounter: CTU;
	testreset: BOOL;
	bConeFeedConvRst: BOOL;
	bStopHmitemp: BOOL;
	step3: INT;
	TON_7: TON;
	R_TRIG_4: R_TRIG;
	bAUnitBConeCrossingOff_2: BOOL;
	testCounter_2: CTU;
	i3ConeCountVal: INT;
	CTU_2_UB: CTU;
	i18ConeCountVal: INT;
	bConveyorStarted: BOOL;
	bConePresentInConv_1: BOOL;
	bAAutoRetrivalEnabled: BOOL;
	bStartConeFeedConvInBypass: BOOL;
END_VAR
bQAFeedingConveyorMotor:=(bAConveStartsAuto);



IF bAutoModeOn AND NOT  bIMCStop  THEN
AllOutputsOn:=TRUE;
ELSE
AllOutputsOn:=FALSE;
END_IF

IF AllOutputsOn AND NOT bIConeOrientationTop AND bIConeFeedingPistonHome  AND NOT bAPauseSeq AND bAMcStartInAuto  THEN
bAConveStartsAuto:=TRUE;
ELSE
bAConveStartsAuto:=FALSE;

END_IF


(*
CASE step2 OF

	0:	R_TRIG_3(CLK:=bIUnitAConeCrossing , Q=> );
		IF R_TRIG_3.Q THEN TON_6(IN:= FALSE); step2:=step2+1; END_IF


	1:	TON_6(IN:= FALSE);
		step2:=step2+1;


	2:	 bAUnitBConeCrossing_1 :=TRUE;
		 step2:=6;

	3:	 step2:=step2+1;

	4: 	TON_6(IN:=  TRUE  , PT:=t#1ms , Q=> , ET=> );
		IF TON_6.Q THEN  step2:=step2+1; END_IF


	5:	 step2:=step2+1;

	6:	bAUnitBConeCrossingOff:=TRUE;
		TON_6(IN:= FALSE);
		step2:=step2+1;

	7:	 step2:=step2+1;

	8:	IF bAUnitBConeCrossingOff THEN bAUnitBConeCrossing_1:=FALSE; step2:=step2+1; END_IF

	9:	 step2:=step2+1;

	10:	bAUnitBConeCrossingOff:=FALSE;
		step2:=0;


END_CASE




*)


testCounter(
	CU:= bIUnitBConeCrossing,
	RESET:= ,
	PV:= ,
	Q=> ,
	CV=> );



(*===============Stop Sequence===========*)


IF NOT  bIEmergency OR bStopHmi  OR bAutoModeOff OR bIMCStop  THEN
	bConeFeedConvRst:=TRUE;
	bAMcStartInAuto:=FALSE;
	testCounter.RESET:=TRUE;
	bInterlockInitial_2:=FALSE;
 ELSE
	bConeFeedConvRst:=FALSE;
	testCounter.RESET:=FALSE;
	END_IF


IF bConeFeedConvRst THEN

bAConveStartsAuto:=FALSE;
END_IF



(*==================Logic is to Run the ConeFeed Conveyor Witout Retreival Unit===============*)

IF NOT bAAutoRetrivalEnabled AND bAutoModeOn AND bIMcStart  THEN bStartConeFeedConvInBypass:=TRUE; ELSE bStartConeFeedConvInBypass:=FALSE; END_IF


(*==========All Outputs Off whenchange l mode to manual  from Auto maode==========*)
END_PROGRAM

(* POU Serial, ST *)
PROGRAM Serial
VAR
	bSendStr:BOOL;
	Timer: TON;
	TrigSend:R_TRIG;
	(*TransmitStr : SendString;*)
	SendBusy: BOOL;
	SendErrorID: ComError_t;

	(*ReceiveStr :ReceiveString;*)
	ReStr: STRING;
	LastReceivedString: STRING;
	StringReceived: BOOL;
	ReceiveBusy: BOOL;
	ReceiveError: BOOL;
	ReceiveErrorID: ComError_t;
	ReceiveTimeout: BOOL;
	ReceiveCounter: UDINT;

	(* Serial communication with the COM port device *)
	(*COMportControl: SerialLineControl;*)
	COMportControlError: BOOL;
	COMportControlErrorID: ComError_t;


	Decimaldata: BYTE;
	Stringdata: STRING;
	RxBufferStringdata: STRING(300);
	TxBufferStringdata: STRING(300);
	RxBufferArrdata: ARRAY [0..80] OF BYTE;
	TxBufferArrdata: ARRAY [0..80] OF BYTE :=(*16#0F, 16#FA, 16#03, 16#00, 16#0D, 16#00, 16#10, 16#20, 16#01, 16#05, 16#58, 16#DF, 16#98, 16#00, 16#00, 16#02, 16#04, 16#E0, 16#B4, 16#F0;*)
16#0F, 16#FA, 16#03, 16#00, 16#02, 16#00, 16#38, 16#24, 16#F0; (*16#00, 16#00, 16#00, 16#00;, 16#10, 16#20, 16#05, 16#02, 16#AF, 16#F6, 16#98, 16#00, 16#00, 16#02, 16#04, 16#E0, 16#84, 16#F0;*)
	i: INT;
	(*ReceiveData_1: ReceiveData;*)

	SReceivedataFormat: ARRAY [0..300] OF BYTE;
	SReceivedatStringFt: STRING(300);
	sSendString_1: STRING(300);
	(*TransmitArrByteData: SendData;*)
(*==============port 2==========*)
	(*ReceiveData_2: ReceiveData;*)

	test: BOOL;
	SReceivedataFormat_2: ARRAY [0..300] OF BYTE;
	SReceivedatStringFt_2: STRING(300);
	(*COMportControl_2: SerialLineControl;*)
	COMportControlError_2: BOOL;
	COMportControlErrorID_2: ComError_t;
	SReceivedatStringFtTemp: STRING;
	SReceivedatStringFt_2Temp: STRING(80);
	(*ReceiveData_3: ReceiveData;*)
	SReceivedataFormat_3: ARRAY [0..300] OF BYTE;
	SReceivedatStringFt_3: STRING(300);
	SReceivedatStringFt_3Temp: STRING;
	(*COMportControl_3: SerialLineControl;*)
	COMportControlError_3: BOOL;
	COMportControlErrorID_3: ComError_t;
	(*ReceiveByte_2: ReceiveByte;*)
	(*ModbusRtuMaster_KL6x22B_3: ModbusRtuMaster_KL6x22B;*)
	ModbusRtuMaster_KL6x22B_3: ModbusRtuMaster_KL6x22B;
	ModbusRtuMaster_KL6x22B_4: ModbusRtuMaster_KL6x22B;
	step1: INT;
	TON1: TON;

	TON_2: TON;
	bUnitARead: BOOL;
	bUnitAreadOk: BOOL;
	bUnitBreadOk: BOOL;
	bUnitBRead: BOOL;

	step2: INT;
	GrossWeightRead: BOOL;
	TON1Gross: TON;
	TON_2Gross: TON;




	resultWt_1: STRING;
	ReceiveString_sample_1: ReceiveString;
	ipos_1: INT;
	prefix_data_1: BYTE ;
	sufix_data_1: BYTE;
	samplestring_1: STRING;

	resultWt_2: STRING;
	ReceiveString_sample_2: ReceiveString;
	ipos_2: INT;
	prefix_data_2: BYTE ;
	sufix_data_2: BYTE;
	samplestring_2: STRING;
END_VAR
ModbusRtuMaster_KL6x22B_3.ReadInputRegs(*ModbusRtuMaster_KL6x22B_3.ReadRegs*)(

	UnitID:=liD ,
	Quantity:=QTY ,
	MBAddr:=IADD ,
	cbLength:=SIZEOF(SReceiveData) ,
	pMemoryAddr:=ADR(SReceiveData) ,
	Execute:=ModbusRead ,
	Timeout:=t#5s ,
	BUSY=>ModBusBussy ,
	Error=>bAModBusError,
	ErrorId=> ,
	cbRead=> );

ModbusRtuMaster_KL6x22B_4.ReadInputRegs(*ModbusRtuMaster_KL6x22B_4.ReadRegs*)(

	UnitID:=liDGross ,
	Quantity:=QTYGross ,
	MBAddr:=IADDGross ,
	cbLength:=SIZEOF(SReceiveDataGross) ,
	pMemoryAddr:=ADR(SReceiveDataGross) ,
	Execute:=ModbusReadGross ,
	Timeout:=t#5s ,
	BUSY=>ModBusBussyGross ,
	Error=>bAModBusErrorGross,
	ErrorId=> ,
	cbRead=> );

(****************
CASE step1 OF


0:	IF  bInterlockInitial_2 AND NOT bUnitARead AND (bUnitBRead OR bUnitBReadInt) AND NOT ModBusBussy THEN bUnitAreadOk:=TRUE;bUnitBreadOk:=FALSE;step1:=step1+1;
	ELSIF bInterlockInitial_2 AND bUnitARead AND  NOT bUnitBRead AND NOT ModBusBussy  THEN bUnitAreadOk:=FALSE;bUnitBreadOk:=TRUE;step1:=step1+1;END_IF


1:	bUnitBReadInt:=FALSE;TON1(IN:=FALSE);TON_2(IN:=FALSE);step1:=step1+1;

2:	IF   bUnitAreadOk AND NOT  ModBusBussy  THEN liD:=1;QTY:=2;IADD:=3;step1:=step1+1;
	ELSIF  bUnitBreadOk AND NOT  ModBusBussy  THEN liD:=2;QTY:=2;IADD:=3;step1:=step1+1;
	END_IF


3:	ModbusRead:=TRUE;
	TON1(IN:=TRUE , PT:= t#0.3s, Q=> , ET=> );
	IF TON1.Q THEN
	step1:=step1+1;
	END_IF

4:	VAR_6:=100;
	VAR_111:=SReceiveData[1];step1:=step1+1;

5:	 IF VAR_111 > 0  THEN VAR_8:=(VAR_111  /  VAR_6);step1:=step1+2;
	ELSIF  VAR_111 = 0 THEN VAR_8:=0;ModbusRead:=FALSE; step1:=step1+1;END_IF

6:	step1:=step1+1;

7:	ModbusRead:=FALSE;
	IF   bUnitAreadOk THEN  rRetUnitAWeight:=VAR_8;step1:=step1+1;
	ELSIF  bUnitBreadOk THEN  rRetUnitBWeight:=VAR_8;step1:=step1+1;END_IF



8:	TON_2(IN:=TRUE , PT:=t#1s , Q=> , ET=> );
	IF TON_2.Q THEN step1:=step1+1;END_IF

9:	IF bUnitAreadOk THEN bUnitARead:=TRUE;bUnitBRead:=FALSE;step1:=0;
	ELSIF bUnitBreadOk THEN bUnitARead:=FALSE;bUnitBRead:=TRUE;step1:=0;END_IF

END_CASE*******************)



CASE step1 OF


0:	IF  bInterlockInitial_2 AND NOT bUnitARead AND (bUnitBRead OR bUnitBReadInt) AND NOT ModBusBussy THEN bUnitAreadOk:=TRUE;bUnitBreadOk:=FALSE;step1:=step1+1;
	ELSIF bInterlockInitial_2 AND bUnitARead AND  NOT bUnitBRead AND NOT ModBusBussy  THEN bUnitAreadOk:=FALSE;bUnitBreadOk:=TRUE;step1:=step1+1;END_IF


1:	bUnitBReadInt:=FALSE;TON1(IN:=FALSE);TON_2(IN:=FALSE);step1:=step1+1;

2:	IF   bUnitAreadOk AND NOT  ModBusBussy  THEN liD:=1;QTY:=2;IADD:=3;step1:=step1+1;
	ELSIF  bUnitBreadOk AND NOT  ModBusBussy  THEN liD:=2;QTY:=2;IADD:=3;step1:=step1+1;
	END_IF


3:	ModbusRead:=TRUE;
	TON1(IN:=TRUE , PT:= t#0.3s, Q=> , ET=> );
	IF TON1.Q THEN
	step1:=step1+1;
	END_IF

4:	VAR_115:=256;VAR_6:=1000;
	  VAR_111:=SReceiveData[1];VAR_2:=SReceiveData[2];VAR_10:=SReceiveData[4];step1:=step1+1;

5:	IF SReceiveData[4]=1 THEN VAR_11:=65536;step1:=step1+1;
	ELSIF SReceiveData[4]=0 THEN VAR_11:=0; step1:=step1+1;END_IF

6:
	VAR_3:=BYTE_TO_REAL(VAR_111) *  (VAR_115);
	VAR_4:=(VAR_3 + VAR_11 + BYTE_TO_REAL(VAR_2));
	step1:=step1+1;

7:	 IF VAR_4 > 0  THEN VAR_8:=(VAR_4  /  VAR_6);step1:=step1+2;
	ELSIF  VAR_4 = 0 THEN VAR_8:=0;ModbusRead:=FALSE; step1:=step1+1;END_IF

8:	step1:=step1+1;



9:	ModbusRead:=FALSE;
	IF   bUnitAreadOk THEN  rRetUnitAWeight:=VAR_8;step1:=step1+1;
	ELSIF  bUnitBreadOk THEN  rRetUnitBWeight:=VAR_8;step1:=step1+1;END_IF



10:	TON_2(IN:=TRUE , PT:=t#0.5s , Q=> , ET=> );
	IF TON_2.Q THEN step1:=step1+1;END_IF

11:	IF bUnitAreadOk THEN bUnitARead:=TRUE;bUnitBRead:=FALSE;step1:=0;
	ELSIF bUnitBreadOk THEN bUnitARead:=FALSE;bUnitBRead:=TRUE;step1:=0;END_IF

END_CASE







CASE step2 OF


0:	IF  bInterlockInitial_2 AND   NOT ModbusReadGross THEN step2:=1;
	END_IF


1:	TON1Gross(IN:=FALSE);TON_2Gross(IN:=FALSE);step2:=2;

2:	IF   NOT  ModBusBussyGross  THEN liDGross:=4;QTYGross:=2;IADDGross:=3;step2:=3;
	END_IF


3:	ModbusReadGross:=TRUE;
	TON1Gross(IN:=TRUE , PT:= t#0.5s, Q=> , ET=> );
	IF TON1Gross.Q THEN
	step2:=4;
	END_IF

4:	TON1Gross(IN:=FALSE);
	VAR_115Gross:=256;VAR_6Gross:=1000;
	  VAR_111Gross:=SReceiveDataGross[1];VAR_2Gross:=SReceiveDataGross[2];VAR_10Gross:=SReceiveDataGross[4];step2:=5;

5:	IF SReceiveDataGross[4]=1 THEN VAR_11Gross:=65536;step2:=6;
	ELSIF SReceiveDataGross[4]=0 THEN VAR_11Gross:=0; step2:=6;END_IF
6:
	VAR_3Gross:=BYTE_TO_REAL(VAR_111Gross) *  (VAR_115Gross);
	VAR_4Gross:=(VAR_3Gross + VAR_11Gross + BYTE_TO_REAL(VAR_2Gross));
	step2:=7;

7:	 IF VAR_4Gross > 0  THEN VAR_8Gross:=(VAR_4Gross  /  VAR_6Gross);step2:=9;
	ELSIF  VAR_4Gross = 0 THEN VAR_8Gross:=0;ModbusReadGross:=FALSE; step2:=9;END_IF

8:	step2:=step2+1;



9:	ModbusReadGross:=FALSE;
	  rGrossWeight:=VAR_8Gross;step2:=10;




10:	TON_2Gross(IN:=TRUE , PT:=t#0.5s , Q=> , ET=> );
	IF TON_2Gross.Q THEN step2:=11;END_IF

11:	step2:=0;


END_CASE


(*==============El6002 serial Communication Program for Laod Cell value read in Rs232 port 1 ==================*)


COMportControl(
	Mode:= SERIALLINEMODE_EL6_22B,
	pComIn:= ADR(COMin_COMport),
	pComOut:= ADR(COMout_COMport),
	SizeComIn:= SIZEOF(COMin_COMport),
	TxBuffer:= TxBuffer1,
	RxBuffer:= RxBuffer1,
	Error=> COMportControlError,
	ErrorID=> COMportControlErrorID );



ReceiveString_sample_1(
	Prefix:='w' ,
	Suffix:='g' ,
	Timeout:= t#5s,
	Reset:= ,
	ReceivedString:=samplestring_1 ,
	RXbuffer:= RxBuffer1,
	StringReceived=> ,
	Busy=> ,
	Error=> ,
	RxTimeout=> );
ipos_1:=FIND(samplestring_1,'n');

resultWt_1:= MID (samplestring_1,9,ipos_1+1);

(*RetWeight*)rRetUnitAWeight:=STRING_TO_REAL(resultWt_1);

(************************************
MAIN.string_Dec();

***)



(*
FOR i:=0 TO 300 DO
	RxBufferStringData[i]:= RxBuffer1.Buffer[i];
END_FOR*)
(**************************************
ReceiveData_1(
	pPrefix:= ,
	LenPrefix:= ,
	pSuffix:= ,
	LenSuffix:= ,
	pReceiveData:=  ADR(SReceivedataFormat),
	SizeReceiveData:= 100,
	Timeout:=t#1s ,
	Reset:= ,
	RXbuffer:=RxBuffer1 ,
	DataReceived=> ,
	busy=> ,
	Error=> ,
	RxTimeout=> ,
	LenReceiveData=> );

MEMCPY(ADR(SReceivedatStringFt), ADR(SReceivedataFormat), 50);

SReceivedatStringFtTemp:=MID(STR:=SReceivedatStringFt, LEN:=7, POS:=3);


 rRetUnitAWeight:=STRING_TO_REAL (SReceivedatStringFtTemp);******************************)

(*==============El6002 serial Communication Program for Laod Cell value read in Rs232 port 2 ==================*)

COMportControl_2(
	Mode:= SERIALLINEMODE_EL6_22B,
	pComIn:= ADR(COMin_2_COMport_2),
	pComOut:= ADR(COMout_2_COMport_2),
	SizeComIn:= SIZEOF(COMin_2_COMport_2),
	TxBuffer:= TxBuffer2,
	RxBuffer:= RxBuffer2,
	Error=> COMportControlError_2,
	ErrorID=> COMportControlErrorID_2 );




ReceiveString_sample_2(
	Prefix:='w' ,
	Suffix:='g' ,
	Timeout:= t#5s,
	Reset:= ,
	ReceivedString:=samplestring_2 ,
	RXbuffer:= RxBuffer2,
	StringReceived=> ,
	Busy=> ,
	Error=> ,
	RxTimeout=> );
ipos_2:=FIND(samplestring_2,'n');

resultWt_2:= MID (samplestring_2,9,ipos_1+1);

(*RetWeight*)rRetUnitBWeight:=STRING_TO_REAL(resultWt_2);


(***************************************
ReceiveData_2(
	pPrefix:= ,
	LenPrefix:= ,
	pSuffix:= ,
	LenSuffix:= ,
	pReceiveData:=  ADR(SReceivedataFormat_2),
	SizeReceiveData:= 100,
	Timeout:=t#1s ,
	Reset:= ,
	RXbuffer:=RxBuffer2 ,
	DataReceived=> ,
	busy=> ,
	Error=> ,
	RxTimeout=> ,
	LenReceiveData=> );

MEMCPY(ADR(SReceivedatStringFt_2), ADR(SReceivedataFormat_2), 50);

 rRetUnitBWeight:=STRING_TO_REAL (SReceivedatStringFt_2);


SReceivedatStringFt_2Temp:=MID(STR:=SReceivedatStringFt_2, LEN:=7, POS:=3);


 rRetUnitBWeight:=STRING_TO_REAL (SReceivedatStringFt_2Temp);*******************************)



(*==============El6002 serial Communication Program for Laod Cell value read in Rs232 port 2 (  GROSS WEIGHT    )  ==================*)

COMportControl_3(
	Mode:= SERIALLINEMODE_EL6_22B,
	pComIn:= ADR(COMin_3_COMport_3),
	pComOut:= ADR(COMout_3_COMport_3),
	SizeComIn:= SIZEOF(COMin_3_COMport_3),
	TxBuffer:= TxBuffer3,
	RxBuffer:= RxBuffer3,
	Error=> COMportControlError_3,
	ErrorID=> COMportControlErrorID_3 );





(******************************
ReceiveData_3(
	pPrefix:= ,
	LenPrefix:= ,
	pSuffix:= ,
	LenSuffix:= ,
	pReceiveData:=  ADR(SReceivedataFormat_3),
	SizeReceiveData:= 100,
	Timeout:=t#1s ,
	Reset:= ,
	RXbuffer:=RxBuffer3 ,
	DataReceived=> ,
	busy=> ,
	Error=> ,
	RxTimeout=> ,
	LenReceiveData=> );

MEMCPY(ADR(SReceivedatStringFt_3), ADR(SReceivedataFormat_3), 50);




SReceivedatStringFt_3Temp:=MID(STR:=SReceivedatStringFt_3, LEN:=7, POS:=3);


 rGrossWeight:=STRING_TO_REAL (SReceivedatStringFt_3Temp);


*)

(*
ReceiveByte_2(
	RxBuffer:=  RxBuffer2  ,
	ByteReceived=> ,
	ReceivedByte=> ,
	Error=> );


*)
(*************CASE step1 OF


0:	IF    NOT ModBusBussy THEN step1:=step1+1;END_IF


1:	TON1(IN:=FALSE);TON_2(IN:=FALSE);step1:=step1+1;

2:	IF   NOT  ModBusBussy  THEN liD:=1;QTY:=2;IADD:=3;step1:=step1+1;
	END_IF


3:	ModbusRead:=TRUE;
	TON1(IN:=TRUE , PT:= t#0.1s, Q=> , ET=> );
	IF TON1.Q THEN
	step1:=step1+1;
	END_IF

4:	VAR_115:=256;VAR_6:=1000;
	  VAR_111:=SReceiveData[1];VAR_2:=SReceiveData[2];VAR_10:=SReceiveData[4];step1:=step1+1;

5:	IF SReceiveData[4]=1 THEN VAR_11:=65536;step1:=step1+1;
	ELSIF SReceiveData[4]=0 THEN VAR_11:=0; step1:=step1+1;END_IF

6:
	VAR_3:=BYTE_TO_REAL(VAR_111) *  (VAR_115);
	VAR_4:=(VAR_3 + VAR_11 + BYTE_TO_REAL(VAR_2));
	step1:=step1+1;

7:	 IF VAR_4 > 0  THEN VAR_8:=(VAR_4  /  VAR_6);step1:=step1+2;
	ELSIF  VAR_4 = 0 THEN VAR_8:=0;ModbusRead:=FALSE; step1:=0;END_IF

8:	step1:=step1+1;



9:	ModbusRead:=FALSE; Ret_ActWt:=VAR_8;step1:=step1+1;



10:	TON_2(IN:=TRUE , PT:=t#1s , Q=> , ET=> );
	IF TON_2.Q THEN step1:=0;END_IF

END_CASE**************)
END_PROGRAM

(* POU AutoMode/FwdPiston, ST *)
PROGRAM FwdPiston
VAR
	step: INT;
	bA2ndConeReached: BOOL;
	bA3rdConeReached: BOOL;
	bAFirstConeReached: BOOL;


	InterLockCounter: CTU;
	R_TRIG_1: R_TRIG;
	step2: INT;
	bAFwdPistonReady: BOOL;


	TimerON: TON;
	R_TRIG_2: R_TRIG;
	bWrapConvStarted: BOOL;
	F_TRIG_1: F_TRIG;
	bConutEnable: BOOL;
	bA3Pushed: BOOL;
	Step12: INT;
	R_TRIG_5: R_TRIG;
	TON_5: TON;
END_VAR
	(*=============================Forward piston On/Off logic =======================*)


CASE step OF


	0:	IF  bAFwdPistonReady AND  bAConeFeedOver   THEN
		bAFirstConeReached:=TRUE;
		InterLockCounter.RESET:=TRUE;
		step:=step+1;
		END_IF

	1:	IF NOT bAPauseSeq THEN InterLockCounter.RESET:=FALSE ;step:=step+1; END_IF

	2:	IF  NOT bQAWrappingConveyorMotor  AND bAutoModeOn  AND bAFirstConeReached    AND InterLockCounter.CV=0(*  AND Wrapping_Unit.bA3Pushed  *)
		AND NOT bAConeMissErrorAtWrpConv  AND NOT bConeMiss2AtWrapConv THEN
		bQAForwardPistonValve:=TRUE;
		 bAErrorChkBit:=TRUE;
		bAConeFeedOver:=FALSE;
		step:=step+1;
		END_IF

	3:	IF NOT bAPauseSeq THEN step:=step+1; END_IF

	4:	IF  bAutoModeOn AND bIForwardPistonEnd AND NOT bAFwdCylRsError  THEN

		(*bQAForwardPistonValve:=FALSE; *)
		bAFirstConeReached:=FALSE;

		bAFwdPistonComp1:=TRUE;
		step:=step+1;
		END_IF

